METHOD Blink
VAR 
	i : INT;
END_VAR
_toggle(inOffTime:=inBlinkPeriod,inOnTime:=inBlinkPeriod);
_heartBeat := _toggle.IsOn;

FOR i := 0 TO LAST_ICON_INDEX DO
	IF _iconSet[i].BlinkingEnabled AND NOT _iconSet[i].Signal THEN 
		_iconSet[i].SignalBlink := _toggle.IsOn;		
	ELSE
		_iconSet[i].SignalBlink := _iconSet[i].Signal;
	END_IF
END_FOR
END_METHOD

METHOD Clear
_iconSet := _iconSetClear;
_badgeValue := 0;
_currentIndex := 0;
END_METHOD

METHOD CountSignals
VAR
	_iconIndex : INT;
END_VAR
_iconIndex := 0;
_badgeValue := 0;
FOR _iconIndex := 0 TO LAST_ICON_INDEX DO
	IF _iconSet[_iconIndex].Title <> '' AND  _iconSet[_iconIndex].EnableRedIcon THEN 
		_badgeValue := _badgeValue + BOOL_TO_INT(NOT _iconSet[_iconIndex].Signal);
	END_IF
END_FOR
END_METHOD

METHOD SetSignal
VAR_INPUT
	inTitle : STRING;
	inSignal : BOOL;
END_VAR

VAR
	_index : INT;
END_VAR
FOR _index := 0 TO LAST_ICON_INDEX DO 
	IF _iconSet[_index].Title = inTitle THEN 
		_iconSet[_index].Signal := inSignal;
		RETURN;
	END_IF
END_FOR
END_METHOD

END_FUNCTION_BLOCK

// ---- Abstractions/CUBase/Tasks/CUBaseAutomat.TcPOU
FUNCTION_BLOCK ABSTRACT CUBaseAutomat EXTENDS TcoTaskedSequencer
VAR
    _dialog : TcoCore.TcoDialog(THIS^);
    _dialogCustomized : TcoCore.TcoCustomizedDialog(THIS^);
    _dialogWithInput : TcoCore.TcoInputDialog(THIS^);
    {attribute addProperty Name "<#Clear counter#>"}
    _counterDataClear : TcoCore.TcoTask(THIS^);
END_VAR
VAR PERSISTENT
    _counterData : BasicCounterData := (Parent := THIS^);
END_VAR

METHOD PUBLIC ClearCounter
VAR_INPUT
END_VAR
_counterData.Passed := 0;
_counterData.Failed := 0;


_counterData.Total := _counterData.Passed + _counterData.Failed;
END_METHOD

PROPERTY PUBLIC ClearCounterDataTask : REFERENCE TO TcoCore.TcoTask
GET
ClearCounterDataTask ref=_counterDataClear;
END_GET
END_PROPERTY

METHOD Count
VAR_INPUT
	Header 		: EntityHeader;
	
END_VAR


IF NOT Header.IsEmpty THEN

    _counterData.LifeTime := _counterData.LifeTime + 1;

    IF Header.Results.Result = eOverallResult.Failed THEN
        _counterData.Failed := _counterData.Failed + 1;
        _counterData.LifeTimeFailed := _counterData.LifeTimeFailed + 1;
    ELSE
        _counterData.Passed := _counterData.Passed + 1;
        _counterData.LifeTimePassed := _counterData.LifeTimePassed + 1;
    END_IF

END_IF;

_counterData.Total := _counterData.Passed + _counterData.Failed;
END_METHOD

(*~
	<docu>
		<summary>
			Stores the data from this controlled unit into the repository. In addition modifies entity header and controlled unit header.									
		</summary>
	</docu>
~*)
METHOD DataEntityClose
VAR_INPUT
	(*~
	<docu>
		<summary>
			The unique step id definition.
		</summary>			
	</docu>	
	~*)
	inStepID : INT;
	(*~
	<docu>
		<summary>
			If input enum is set to InvokeAndWaitDone  operation will  wait until task reaches the ```Done``` state .
			If input enum is set to InvokeOnly results return True when  task reaches the ```Busy``` state . Later is recomended (neccessary) to check  task  ```Done``` state  , check  task  status.
		</summary>			
	</docu>	
	~*)
	InvokeAction: eDataEntityInvokeType;
END_VAR
VAR_IN_OUT
	Header : CuHeader; 
END_VAR
IF (Step(inStepID,TRUE, 'CLOSE ENTITY DATA')) THEN
    //-------------------------------------		
	IF IsFreshState THEN
		Count(THIS^.StationBase.ProcessDataManager.Data.EntityHeader);
	END_IF
	CASE InvokeAction OF
		eDataEntityInvokeType.InvokeAndWaitDone: 
				StepCompleteWhen(THIS^.StationBase.EntityFlowCloseForOperations(Header).Done);
		eDataEntityInvokeType.InvokeOnly: 
				StepCompleteWhen(THIS^.StationBase.EntityFlowCloseForOperations(Header).Busy);	
	END_CASE;			   		    				
    //-------------------------------------
END_IF
END_METHOD

(*~
	<docu>
		<summary>
			Creates new record in the repository with given EntityId and populates with the current controlled units data.
			In addition modifies entity header and controlled unit header.									
		</summary>
	</docu>
~*)
METHOD DataEntityCreateNew
VAR_INPUT	
	inStepID : INT;
	EntityId : STRING(255);
END_VAR

VAR_IN_OUT
	Header: CuHeader;
END_VAR
IF (Step(inStepID, TRUE, 'CREATE NEW ENTITY DATA')) THEN
    //-------------------------------------		
	StepCompleteWhen(THIS^.StationBase.EntityFlowCreateNew(EntityId, Header).Done);				   		    				
    //-------------------------------------
END_IF
END_METHOD

METHOD DataEntityDiscard
VAR_INPUT	
	inStepID : INT;
	EntityId : STRING(255);
END_VAR
VAR_IN_OUT
	Header: CuHeader;
END_VAR
IF (Step(inStepID, TRUE, 'DISCARD ENTITY DATA')) THEN
    //-------------------------------------		
	StepCompleteWhen(THIS^.StationBase.EntityFlowDiscard(EntityId, Header).Done);				   		    				
    //-------------------------------------
END_IF
END_METHOD

(*~
	<docu>
		<summary>
			Stores data of this controlled unit into the repository.
			In addition modifies entity header and controlled unit header.
			Finalize will set the comprehensive result from InProgress to Passed. 
			If the comprehensive result is Failed the finalizing will not modify the result.									
		</summary>
	</docu>
~*)
METHOD DataEntityFinalize : BOOL
VAR_INPUT
	(*~
	<docu>
		<summary>
			The unique step id definition.
		</summary>			
	</docu>	
	~*)
	inStepID : INT;
	(*~
	<docu>
		<summary>
			If input enum is set to InvokeAndWaitDone  operation will  wait until task reaches the ```Done``` state .
			If input enum is set to InvokeOnly results return True when  task reaches the ```Busy``` state . This option is used when we need to reduce cycle time. Later is recomended (neccessary) to check  task  ```Done``` state  , check  task  status.
		</summary>			
	</docu>	
	~*)
	InvokeAction: eDataEntityInvokeType;
END_VAR
VAR_IN_OUT
	Header: CuHeader;
END_VAR
IF (Step(inStepID,TRUE, 'FINALIZE ENTITY DATA')) THEN
    //-------------------------------------		
		CASE InvokeAction OF
		eDataEntityInvokeType.InvokeAndWaitDone: 
				StepCompleteWhen(THIS^.StationBase.EntityFlowFinalize(Header).Done);
		eDataEntityInvokeType.InvokeOnly: 
				StepCompleteWhen(THIS^.StationBase.EntityFlowFinalize(Header).Busy);	
	END_CASE;			   		    				
		   		    				
    //-------------------------------------
END_IF
END_METHOD

(*~
	<docu>
		<summary>
			Retrieves the data with given EntityId from the repository. In addition modifies entity header and controlled unit header.									
		</summary>
	</docu>
~*)
METHOD DataEntityOpen
VAR_INPUT
	(*~
	<docu>
		<summary>
			The unique step id definition.
		</summary>			
	</docu>	
	~*)
	inStepID : INT;
	(*~
	<docu>
		<summary>
			The definition of jump sptep.Usage of this jump step is when entity does not belong to the Controled unit.
		</summary>			
	</docu>	
	~*)
	inReqStepId: INT;
	inEntityId : STRING(255);
END_VAR
VAR_IN_OUT
	CuHeader: CuHeader;
END_VAR
IF (Step(inStepID, TRUE, 'OPEN ENTITY DATA')) THEN
    //-------------------------------------		
    IF THIS^.StationBase.EntityFlowOpenForOperations(inEntityId, CuHeader).Done THEN
        IF THIS^.StationBase.ProcessDataManager.Data.EntityHeader.IsEmpty THEN
            RequestStep(inReqStepId);
        ELSIF EntityDoesBelong() THEN
            CompleteStep();
        ELSE
            RequestStep(inReqStepId);
        END_IF
    END_IF;
    //-------------------------------------
END_IF
END_METHOD

METHOD EntityDoesBelong : BOOL
VAR_INPUT
END_VAR
EntityDoesBelong:=THIS^.StationBase.ProcessDataManager.Data.EntityHeader.NextStation = THIS^.StationBase.CuId;
END_METHOD

METHOD PUBLIC  HideAllDialogs
VAR_INPUT
END_VAR
_dialog.Restore();
_dialogWithInput.Restore();
_dialogCustomized.Restore();
END_METHOD

METHOD MonitorAnyRecurringFailure
VAR_INPUT
	(*~
	<docu>
		<summary>
			The unique step id definition.
		</summary>			
	</docu>	
	~*)
	inStepID : INT;
	(*~
	<docu>
		<summary>
			The step enable condition.
		</summary>			
	</docu>	
	~*)
	inEnableStep :BOOL;
	inResult : TcoComprehensiveResult;
END_VAR
IF (Step(inStepID,inEnableStep, 'MONITOR ANY RECURRING FAILURE IN SEQUENCE')) THEN
    //-------------------------------------		
	
	IF(inResult.Result<>eOverallResult.Failed ) THEN
		THIS^.StationBase.RecurringFails.AnyRecurringFails.Counter:=0;
		THIS^.StationBase.RecurringFails.AnyRecurringFails.Reached :=FALSE;
		This^.CompleteStep();
	ELSE
		//collect any recurring fails
		IF NOT THIS^.StationBase.RecurringFails.AnyRecurringFails.Reached THEN 
			THIS^.StationBase.RecurringFails.AnyRecurringFails.Counter := THIS^.StationBase.RecurringFails.AnyRecurringFails.Counter +1;
		END_IF
		THIS^.StationBase.RecurringFails.AnyRecurringFails.Reached:=THIS^.StationBase.RecurringFails.AnyRecurringFails.Counter>=THIS^.StationBase._settings.AnyRecurringFailure;
		

		
	

		
		THIS^.Messenger.OnCondition(THIS^.StationBase.RecurringFails.AnyRecurringFails.Reached)
									   .Build()
									   .Append('(Consecutive failure) The number of any recurring failure count has been reached!')
									   .Append(' Failure code: ')
									   .Append(inResult.ErrorCodes)
  									   .Append(' ')
									   .Append(inResult.Failures)						
									   .As()				   
									   .AsError();
									   
		THIS^.StepCompleteWhen(NOT THIS^.StationBase.RecurringFails.AnyRecurringFails.Reached);			
						   
									   
		IF THIS^.StationBase.RecurringFails.AnyRecurringFails.Reached THEN
			
				
			IF(_dialog.Show()
			   .WithCaption('<#(Consecutive failure) The number of any recurring failure count has been reached!#>')
			   .WithText('<#Please acknowledge recurring failure!#>')
			   .WithOk().Answer = TcoCore.eDialogAnswer.OK) THEN
			   
					THIS^.StationBase.RecurringFails.AnyRecurringFails.Counter:=0;
					THIS^.StationBase.RecurringFails.AnyRecurringFails.Reached :=FALSE;
					THIS^.CompleteStep();
			END_IF; 
		END_IF;
	END_IF;
	

	
	
	
 		    				
    //-------------------------------------
END_IF
END_METHOD

METHOD MonitorSameRecurringFailure
VAR_INPUT
	(*~
	<docu>
		<summary>
			The unique step id definition.
		</summary>			
	</docu>	
	~*)
	inStepID : INT;
		(*~
	<docu>
		<summary>
			The step enable condition.
		</summary>			
	</docu>	
	~*)
	inEnableStep :BOOL;
	inResult : TcoComprehensiveResult;
END_VAR
IF (Step(inStepID,inEnableStep, 'MONITOR SAME RECURRING FAILURE IN SEQUENCE')) THEN
    //-------------------------------------		
	
	IF(inResult.Result<>eOverallResult.Failed ) THEN
		THIS^.StationBase.RecurringFails.SameRecurringFails.Counter:=0;
		THIS^.StationBase.RecurringFails.SameRecurringFails.Reached :=FALSE;
		THIS^.CompleteStep();
	ELSE
	
		//collect same recurring
		IF NOT THIS^.StationBase.RecurringFails.SameRecurringFails.Reached THEN 
			IF THIS^.StationBase.RecurringFails.SameRecurringFails.Result.ErrorCodes = inResult.ErrorCodes AND inResult.ErrorCodes <>';' THEN //if error code not defined ignore
				THIS^.StationBase.RecurringFails.SameRecurringFails.Counter := THIS^.StationBase.RecurringFails.SameRecurringFails.Counter +1;
			END_IF;
			THIS^.StationBase.RecurringFails.SameRecurringFails.Result.ErrorCodes := inResult.ErrorCodes ;
		END_IF;
		
		THIS^.StationBase.RecurringFails.SameRecurringFails.Reached:=THIS^.StationBase.RecurringFails.SameRecurringFails.Counter>=THIS^.StationBase._settings.SameRecurringFailure;

			
		THIS^.Messenger.OnCondition(THIS^.StationBase.RecurringFails.SameRecurringFails.Reached)
									   .Build()
									   .Append('(Consecutive failure) The number of same recurring failure count has been reached!')
									   .Append(' Failure code: ')
									   .Append(inResult.ErrorCodes)
  									   .Append(' ')
									   .Append(inResult.Failures)									   									   
									   .As()				   
									   .AsError();
		
		THIS^.StepCompleteWhen(NOT THIS^.StationBase.RecurringFails.SameRecurringFails.Reached);
	

									   
		IF THIS^.StationBase.RecurringFails.SameRecurringFails.Reached THEN
			IF(_dialog.Show()
			   .WithCaption('<#(Consecutive failure) The number of same recurring failure count has been reached!#>')
			   .WithText('<#Please acknowledge recurring failure!#>')
			   .WithOk().Answer = TcoCore.eDialogAnswer.Ok) THEN
			   
					THIS^.StationBase.RecurringFails.SameRecurringFails.Counter:=0;
					THIS^.StationBase.RecurringFails.SameRecurringFails.Reached :=FALSE;
					THIS^.CompleteStep();
			END_IF; 
		END_IF
	END_IF;
	

	
	
	
 		    				
    //-------------------------------------
END_IF
END_METHOD

PROPERTY StationBase : REFERENCE TO CuBase
GET
VAR
    _station : POINTER TO CUBase;
END_VAR
IF __QUERYPOINTER(Parent, _station) THEN // Check if _Parent is Station001
    StationBase REF= _station^;              // If the check is successful dereference a pointer. simlar to THIS^ or SUPER^
END_IF
END_GET
END_PROPERTY

END_FUNCTION_BLOCK

// ---- Abstractions/TcoCore/TcoTaskedSequencer.TcPOU
FUNCTION_BLOCK PUBLIC ABSTRACT TcoTaskedSequencer EXTENDS TcoCore.TcoSequencerBase
VAR
	{attribute addProperty Name "|[[1]AttributeName]|"}
	{attribute addProperty ToolTip "|[[1]AttributeToolTip]|"}
    _task : TcoInnerTask(THIS^);
    _o    : TcoCore.TcoSequencerObserver(THIS^);	
	
	{attribute addProperty Name "|[[1]Cycle Time Analitics]|"} 
	_cycleTimeAnalitics:CycleTimeAnalitics;	
	_startCleanCycleTime: TIME;
	_stopCleanCycleTime: TIME;
	_timer_1: TON;
	_timer_2: TON;
	_detectStartSeq : R_TRIG;

	_customObserver:TcoCustomSequencerObserver(THIS^);
END_VAR

Run();

PROPERTY PUBLIC AverageCleanCycleTime : TIME
GET
AverageCleanCycleTime:=_cycleTimeAnalitics.AverageCleanCycle;
END_GET
END_PROPERTY

PROPERTY PUBLIC AverageCycleTime : TIME
GET
AverageCycleTime:=_cycleTimeAnalitics.Average;
END_GET
END_PROPERTY

(*~
	<docu>
		<summary>
			Completes the actually running step, when the `inCondition` parameter is `TRUE`.
			Method is typically called inside a step as the transition method.
		</summary>			
	</docu>	
~*)
METHOD PROTECTED FINAL Await
VAR_INPUT
    (*~
	<docu>
		<summary>
			The condition under which the step is completed.
		</summary>			
	</docu>	
~*)
    inCondition : BOOL;
END_VAR
i_StepCompleteWhen(inCondition := inCondition);
END_METHOD

(*~
	<docu>
		<summary>
			<para>
				Completes the sequencer, and return the sequencer pointer to the first step in the seuqence.
				Method is typically called inside the last step of the sequence.
			</para>
		</summary>			
	</docu>	
~*)
METHOD PROTECTED FINAL CompleteSequence



i_CompleteSequence();

IF _cycleTimeAnalitics.FilterConstant = 0 THEN;
	_cycleTimeAnalitics.FilterConstant:=10;
END_IF;


IF _cycleTimeAnalitics.Average = T#0S THEN
	_cycleTimeAnalitics.Average:=_SequenceElapsedTime;
END_IF
_cycleTimeAnalitics.Average:= (((_cycleTimeAnalitics.FilterConstant-1)*_cycleTimeAnalitics.Average)+_LastCycleTime)/_cycleTimeAnalitics.FilterConstant;

_startCleanCycleTime:=T#0S;
_stopCleanCycleTime:=T#0S;
END_METHOD

(*~
	<docu>
		<summary>
			Completes the execution of the current step and moves the sequencer pointer to the next step in order of execution.
			The call returns `ITcoObjectRestorer` that allows to restore object upon step completition.
		</summary>		
		<returns></returns>	
	</docu>	
~*)
METHOD PROTECTED FINAL CompleteStep : ITcoObjectRestorer

CompleteStep := i_CompleteStep();
END_METHOD

PROPERTY CustomObserver : REFERENCE TO TcoCustomSequencerObserver
GET
CustomObserver ref= _customObserver;
END_GET
END_PROPERTY

PROPERTY PUBLIC CycleTimeFilterConstant : UINT
GET
CycleTimeFilterConstant:=_cycleTimeAnalitics.FilterConstant;
END_GET
SET // PUBLIC
_cycleTimeAnalitics.FilterConstant:=CycleTimeFilterConstant;
END_SET
END_PROPERTY

(*~
	<docu>
		<summary>
			Main method of the sequener. Custom code needs to be placed here. The sequencer is executed by call of **Instance.Run()** method.
			This method is abstract, and it must be overridden in derived block.
		</summary>
	</docu>
~*)
METHOD PROTECTED  Main : BOOL
END_METHOD

(*~
	<docu>
		<summary>
			Completes the execution of the current step and moves the sequencer pointer to the next step in order of execution.
			The call returns `ITcoObjectRestorer` that allows to restore object upon step completition.
		</summary>		
		<returns></returns>	
	</docu>	
~*)
METHOD PROTECTED FINAL Next : ITcoObjectRestorer
Next := i_CompleteStep();
END_METHOD

METHOD PUBLIC OnAbort : BOOL
SUPER^.Restore();
END_METHOD

METHOD PUBLIC OnDone : BOOL
END_METHOD

METHOD PUBLIC OnError : BOOL
END_METHOD


(*~
	<docu>
		<summary>
			This method is called on sequence completion (the sequencer's last step was completed). 
			This method can be overridden in derived block with a custom logic.
		</summary>			
	</docu>	
~*)
METHOD PROTECTED OnSequenceCompleted
SUPER^.OnSequenceCompleted();
_customObserver.DefineEndTime(Context.RealTimeClock.NowLocalAsTIMESTRUCT());
_customObserver.CompleteSequence();
END_METHOD

METHOD PUBLIC OnStart
_startCleanCycleTime:=T#0S;
_stopCleanCycleTime:=T#0S;
END_METHOD

(*~
	<docu>
		<summary>
			This method is executed upon step completion.
			This method can be overridden in derived block by custom logic.
		</summary>			
	</docu>	
~*)
METHOD PROTECTED OnStepCompleted


_customObserver.Observe(
	inID:= _currentStep.ID, 
	inDescription:= _currentStep.Description, 
	inDuration:= _currentStep.Duration);
END_METHOD

METHOD pr_Close
VAR_INPUT
END_VAR
_lastClosingCycle := Context.StartCycleCount;

IF _sequencerHasError THEN
    OnSequencerError(_sequencerErrorId);
END_IF

_previousNumberOfStepsInSequence := _numberOfStepsInSequence;
Context.Environment.Messaging.Suspend();

IF _modeController._stepIn.Done THEN
    _modeController._stepIn.Restore();
END_IF

Context.Environment.Messaging.Resume();

_restoringSequence := FALSE;
END_METHOD

METHOD pr_Open
VAR
    _message : STRING(255);
END_VAR
_theOrderOfTheCurrentlyEvaluatedStep := 0;

IF _requestStepActive AND
    _requestedStepId <> (MinStepID - 1) AND
    (_modeController.Mode <> eSequencerMode.StepMode OR _modeController._stepIn.Busy OR _checkStepIdRequestedInStepMode) THEN
    _requestStepCycle := _requestStepCycle + 1;
ELSE
    _requestStepCycle := 0;

END_IF

IF _requestStepCycle > 1 AND NOT _sequencerHasError THEN
    _sequencerErrorId        := eSequencerError.StepWithRequestedIdDoesNotExists;
    _message                 := CONCAT('REQUESTED STEP_ID: ', INT_TO_STRING(_requestedStepId));
    _message                 := CONCAT(_message, ' DOES NOT EXIST');
    _currentStep.Description := _message;
    _currentStep.Status      := eStepStatus.Error;
    THIS^.Messenger.Post(_message, eMessageCategory.ProgrammingError);
    _sequencerHasError := TRUE;

END_IF

IF _StepIdUniquenessControlState = eStepIdUniquenessControlState.NotYetStarted OR
    _StepIdUniquenessControlState = eStepIdUniquenessControlState.Requested THEN
    _StepIdUniquenessControlState := eStepIdUniquenessControlState.Started;

END_IF;

_restoringSequence := FALSE;

_lastOpeningCycle := Context.StartCycleCount;
END_METHOD

(*~
	<docu>
		<summary>
			Terminates the currently executed step and set the sequencer's pointer to the step with Id that corresponds to ```inRequestedStepID``` parameter.
			When the order of the requested step is higher than the order of the currently finished step (the requested step is "after" the current one)
			the requested step is started in the same context cycle.
			When the order of the requested step is lower than the order of the currently finished step (the requested step is "before" the current one)
			the requested step is started in the next context cycle.
			If the requested step is not found even in the next context cycle, the sequencer enters error state ```StepWithRequestedIdDoesNotExists```.
			<para>
				See <see cref="TcoCore.eSequencerError"/> for detailed description.
			</para>
		</summary>
	</docu>
~*)
METHOD PROTECTED FINAL RequestRestoreOrigin : ITcoSequencer

VAR
    _message : STRING(254);
END_VAR
RequestRestoreOrigin := i_RequestStep(inRequestedStepID := RESTORE_STEP_ID);
END_METHOD

(*~
	<docu>
		<summary>
			Terminates the currently executed step and set the sequencer's pointer to the step with Id that corresponds to ```inRequestedStepID``` parameter.
			When the order of the requested step is higher than the order of the currently finished step (the requested step is "after" the current one)
			the requested step is started in the same context cycle.
			When the order of the requested step is lower than the order of the currently finished step (the requested step is "before" the current one)
			the requested step is started in the next context cycle.
			If the requested step is not found even in the next context cycle, the sequencer enters error state ```StepWithRequestedIdDoesNotExists```.
			<para>
				See <see cref="TcoCore.eSequencerError"/> for detailed description.
			</para>
		</summary>
	</docu>
~*)
METHOD PROTECTED FINAL RequestStep : ITcoSequencer
VAR_INPUT
    (*~
		<docu>
			<summary>
				StepId of the step to be executed.
			</summary>
		</docu>
	~*)
    inRequestedStepID : INT := MinStepID - 1;
END_VAR
VAR
    _message : STRING(254);
END_VAR
RequestStep := i_RequestStep(inRequestedStepID := inRequestedStepID);
END_METHOD

(*~
	<docu>
		<summary>
			This method resets the sequencer cycle time . 
				Method is typically called before starting the sequence(e.g.in ground position task) .
		</summary>		
		<returns></returns>	
	</docu>	
~*)
METHOD PUBLIC ResetCycleTime
VAR_INPUT
END_VAR

_cycleTimeAnalitics.Average:=T#0S;
_cycleTimeAnalitics.AverageCleanCycle:=T#0S;
END_METHOD

METHOD PRIVATE ResetTimers
VAR_INPUT
END_VAR
_timer_1.IN:=FALSE;
_timer_2.IN:=FALSE;
END_METHOD

(*~
	<docu>
		<summary>
			<para>
				This method resets the sequencer. 
				Method is typically called before starting the sequence or after error has occured in the sequence.
			</para>
		</summary>			
	</docu>	
~*)
METHOD PUBLIC Restore : ITcoRestorable
SUPER^.Restore();
Task.Restore();
END_METHOD

(*~
	<docu>
		<summary>
			<para>
				Ensures calling the Open(), Main() and Close() methods in the desired order.
				This method is final, so it cannot be overloaded. The **Instance.Run()** needs to be called cyclically inside the appropriate context.
			</para>
		</summary>			
	</docu>	
~*)
METHOD PUBLIC FINAL Run
VAR
    _message : STRING;
END_VAR
IF (_task.Execute()) THEN
    THIS^.pr_Open();

    THIS^.Observer := _o;
    THIS^.Main();
	_detectStartSeq(CLK:=_cycleTimer.ET > T#0S);
    IF _detectStartSeq.Q THEN
        CustomObserver.Clear();
        CustomObserver.DefineStartTime(Context.RealTimeClock.NowLocalAsTIMESTRUCT());
    END_IF

    _customObserver();
    THIS^.pr_Close();
END_IF;
END_METHOD

(*~
	<docu>
		<summary>
			This method s used to start the clean cycle time measurement . 
				Method is typically called at the beggining of the sequence(e.g.in automat sequence) .
		</summary>		
		<returns></returns>	
	</docu>	
~*)

METHOD PUBLIC StartCleanCycleTime
VAR_INPUT
END_VAR
_stopCleanCycleTime:=t#0s;
_startCleanCycleTime:=_SequenceElapsedTime;
END_METHOD

METHOD PROTECTED Step : BOOL
VAR_INPUT
    (*~
	<docu>
		<summary>
			StepId of the current step.
			<remarks>			
				<note type="important">
					This number must be unique throughout the complete sequence.
					It must be a constant or numerical literal and it must not change during the life-time of the sequencer. 
				</note>
			</remarks>
		</summary>		
	</docu>	
~*)
    inStepID : INT;
    (*~
	<docu>
		<summary>
			If this value is false, step body is not executed and execution is moved to the next enabled step.
		</summary>				
	</docu>	
~*)
    inEnabled : BOOL;
    (*~
	<docu>
		<summary>
			Step description text.
		</summary>				
	</docu>	
~*)
    inStepDescription : STRING(254);
END_VAR
Step := i_Step(inStepID := inStepID, inEnabled := inEnabled, inStepDescription := inStepDescription);
END_METHOD

(*~
	<docu>
		<summary>
			Completes the actually running step, when the `inCondition` parameter is `TRUE`.
			Method is typically called inside a step as the transition method.
		</summary>			
	</docu>	
~*)
METHOD PROTECTED FINAL StepCompleteWhen
VAR_INPUT
    (*~
	<docu>
		<summary>
			The condition under which the step is completed.
		</summary>			
	</docu>	
~*)
    inCondition : BOOL;
END_VAR
i_StepCompleteWhen(inCondition := inCondition);
END_METHOD

(*~
	<docu>
		<summary>
			This method s used to stop the clean cycle time measurement . 
				Method is typically called at the end of the sequence(e.g.in automat sequence )  .
		</summary>		
		<returns></returns>	
	</docu>	
~*)

METHOD PUBLIC StopCleanCycleTime
VAR_INPUT
END_VAR

VAR
	cleanCycleTime: TIME;
END_VAR
_stopCleanCycleTime:=_SequenceElapsedTime;

cleanCycleTime:=T#0S;
IF _stopCleanCycleTime>_startCleanCycleTime THEN
	cleanCycleTime:=_stopCleanCycleTime-_startCleanCycleTime;
 END_IF;

IF _cycleTimeAnalitics.FilterConstant = 0 THEN;
	_cycleTimeAnalitics.FilterConstant:=10;
END_IF;


IF _cycleTimeAnalitics.AverageCleanCycle = T#0S THEN
	_cycleTimeAnalitics.AverageCleanCycle:=_stopCleanCycleTime;
END_IF
_cycleTimeAnalitics.AverageCleanCycle:= (((_cycleTimeAnalitics.FilterConstant-1)*_cycleTimeAnalitics.AverageCleanCycle)+cleanCycleTime)/_cycleTimeAnalitics.FilterConstant;
END_METHOD

PROPERTY Task : REFERENCE TO TcoTask
GET
Task REF= _task;
END_GET
END_PROPERTY

METHOD PUBLIC FINAL Timer_1 : BOOL
VAR_INPUT
	Condition : BOOL;
	PT : TIME;
END_VAR
_timer_1(IN:= Condition  and  not IsFreshState, PT:=PT);
Timer_1 := _timer_1.Q;
END_METHOD

METHOD PUBLIC FINAL Timer_2 : BOOL
VAR_INPUT
	Condition : BOOL;
	PT : TIME;
END_VAR
_timer_2(IN:= Condition and not IsFreshState, PT:=PT);
Timer_2 := _timer_2.Q;
END_METHOD

END_FUNCTION_BLOCK

// ---- Abstractions/TcoCore/TcoCustomSequencerObserver.TcPOU
FUNCTION_BLOCK TcoCustomSequencerObserver EXTENDS TcoObject 
VAR
	//~
    _data            : TcoCustomExportSeqData;
	//~
	_dataToExport            : TcoCustomExportSeqData;
	

	_exportSeqData:TcoCore.TcoRemoteTask(THIS^);
	_order:UINT;
END_VAR

VAR CONSTANT
    MAX_STEPS : UINT := 150;
END_VAR

_exportSeqData();

{attribute 'hide'}
METHOD Clear : BOOL
VAR 
	i : INT;
	blank : TcoCustomStepDetails;
END_VAR
{warning disable C0196}
FOR i := 0 TO MAX_STEPS DO
{warning enable C0196}
	_data.Steps[i] := blank;	
END_FOR
_order:=0;
END_METHOD

METHOD CompleteSequence
VAR_INPUT
END_VAR

_dataToExport:=_data;

IF _exportSeqData._isInitialized  THEN
	
	_exportSeqData.Restore();
	_exportSeqData.Invoke();
  
	
END_IF
END_METHOD

METHOD DefineControledUnit
VAR_INPUT
	inCuid: UINT;
END_VAR
_data.CuId:=inCuid;
END_METHOD

METHOD DefineEndTime
VAR_INPUT
	inTime:Tc2_Utilities.TIMESTRUCT;
END_VAR
_data.EndTime.Year :=  inTime.wYear;
_data.EndTime.Month :=  inTime.wMonth;
_data.endTime.Day :=  inTime.wDay;
_data.endTime.Hour :=  inTime.wHour;
_data.endTime.Minute :=  inTime.wMinute;
_data.endTime.Second :=  inTime.wSecond;
_data.endTime.Milliseconds :=  inTime.wMilliseconds;
END_METHOD

METHOD DefineStartTime
VAR_INPUT
	inTime:Tc2_Utilities.TIMESTRUCT;
END_VAR
_data.startTime.Year :=  inTime.wYear;
_data.startTime.Month :=  inTime.wMonth;
_data.startTime.Day :=  inTime.wDay;
_data.startTime.Hour :=  inTime.wHour;
_data.startTime.Minute :=  inTime.wMinute;
_data.startTime.Second :=  inTime.wSecond;
_data.startTime.Milliseconds :=  inTime.wMilliseconds;
END_METHOD

PROPERTY ExportSeqData : REFERENCE TO TcoCore.TcoRemoteTask
GET
ExportSeqData ref=_exportSeqData;
END_GET
END_PROPERTY

(*~
	<docu>
		<summary>
			Provides the mechanism to observe steps in the sequence and to gather basic infomation about step status and perfomance.
		</summary>			
	</docu>	
~*)
METHOD Observe
VAR_INPUT
	
	(*~
	<docu>
		<summary>
			Step identification number.
		</summary>	
		<remarks>			
 			<note type="important">
				This number must be unique throughout the complete sequence. It is required to uniquely identify the step of the sequence.
			</note>
			<para>
				The <see cref="PlcDocu.TcoCore.TcoSequencer.RequestStep"/> method is using this number to jump to the required step.
			</para>
		</remarks>
	</docu>	
	~*)
		{attribute addProperty Name "<#Step ID#>"}
		inID: INT;


	(*~
		<docu>
			<summary>
				Step description text.
			</summary>				
		</docu>	
	~*)
		{attribute addProperty Name "<#Step description#>"}
		inDescription: STRING(254);

	(*~
		<docu>
			<summary>
				Step duration time.
			</summary>				
		</docu>	
	~*)	
		{attribute addProperty Name "<#Step duration#>"}
		inDuration : TIME;	


END_VAR

VAR
	_timeStruct: Tc2_Utilities.TIMESTRUCT;
END_VAR

IF(_order <= MAX_STEPS)  THEN
	_data.Steps[_order].ID := inID;
	_data.Steps[_order].Description := inDescription;
	_data.Steps[_order].Duration := inDuration;
	_timeStruct:=Context.RealTimeClock.NowLocalAsTIMESTRUCT();
	
	_data.Steps[_order].TimeStamp.Year :=  _timeStruct.wYear;
	_data.Steps[_order].TimeStamp.Month :=  _timeStruct.wMonth;
	_data.Steps[_order].TimeStamp.Day :=  _timeStruct.wDay;
	_data.Steps[_order].TimeStamp.Hour :=  _timeStruct.wHour;
	_data.Steps[_order].TimeStamp.Minute :=  _timeStruct.wMinute;
	_data.Steps[_order].TimeStamp.Second :=  _timeStruct.wSecond;
	_data.Steps[_order].TimeStamp.Milliseconds :=  _timeStruct.wMilliseconds;


		
	
	_order:=_order+1;
END_IF;
END_METHOD

METHOD SetCycleId
VAR_INPUT
	inId:string(254);
END_VAR
_data.CycleId:=inId;
END_METHOD

END_FUNCTION_BLOCK

// ---- Abstractions/Generic/LightTower/TcoLightTower.TcPOU
FUNCTION_BLOCK TcoLightTower EXTENDS TcoCore.TcoComponent
VAR_IN_OUT
	{attribute clr [RenderIgnore()]}
	inoGreenLight   :  BOOL;
	
	{attribute clr [RenderIgnore()]}
	inoRedLight     :  BOOL;
	
	{attribute clr [RenderIgnore()]}
	inoOrangeLight  :  BOOL;
	
	{attribute clr [RenderIgnore()]}
	inoBlueLight    :  BOOL;

	{attribute clr [RenderIgnore()]}
	inoHorn         :  BOOL;
END_VAR

VAR
	
	
	{attribute addProperty Name "<#Status#>"}
    {attribute clr [ReadOnly()]}
    _status : TcoLightTower_Status;

	{attribute addProperty Name "<#Config#>"}
    _config : TcoLightTower_Config;
	
    _materrialError : bool;

	//~
	_controlledUnits      : ARRAY [0..12] OF ICUBase;
	//~			
	
	
	// group states

	//~
	{attribute clr [RenderIgnore()]}
	_blinker              : TcoUtilities.TcoBlinker(THIS^);
	{attribute clr [RenderIgnore()]}
	_blinkerSlow              : TcoUtilities.TcoBlinker(THIS^);
	//~

END_VAR

IF _controlledUnits[0] = 0 THEN
    THIS^.Messenger.Programming('<#Missing link to Controlled unit! No function is being executed!#>');
    RETURN;
END_IF

inoGreenLight := FALSE;
inoRedLight := FALSE;
inoOrangeLight := FALSE;
inoBlueLight := FALSE;
inoHorn := FALSE;

_blinker(inOffTime := T#500MS, inOnTime := T#500MS); //2 Hz
_blinkerSlow(inOffTime := T#1250MS, inOnTime := T#1250MS); //0.8 Hz

THIS^.Initialize();

//ground
IF _status.State.AnyGrounding THEN
    inoGreenLight := _blinker.IsOn;
    inoRedLight := _status.State.AnyInError AND _blinker.IsOn;
    inoOrangeLight := _status.State.AnyInWarning AND _blinker.IsOn;
END_IF

//auto
IF _status.State.AllInAuto AND NOT _status.State.AnyInStepMode AND NOT _status.State.AnyInError AND _status.State.AnyInWarning THEN
    inoGreenLight := TRUE; // ok production
ELSIF _status.State.AllInAuto AND _status.State.AnyInStepMode THEN
    inoGreenLight := _blinker.IsOn; //step mode
ELSIF _status.State.AllInAuto AND NOT _status.State.AnyInStepMode THEN
    inoGreenLight := TRUE; // ok production
    inoRedLight := _status.State.AnyInError AND _blinker.IsOn;
    inoOrangeLight := _status.State.AnyInWarning AND _blinker.IsOn;
ELSIF _status.State.AllInManual  THEN

    inoOrangeLight :=  _blinker.IsOn;

END_IF;

IF NOT _config.HornEnabled THEN
    inoHorn := FALSE;
END_IF;

//todo blue should be suitable for material feeding
IF _materrialError AND _status.State.AllInAuto THEN
	inoBlueLight :=  _blinker.IsOn;
END_IF

METHOD AddControlledUnit : BOOL
VAR_INPUT
 	inControlledUnit : ICUBase;
END_VAR
VAR
	i : UINT;
END_VAR
AddControlledUnit := FALSE;

IF inControlledUnit = 0 THEN
	RETURN;
END_IF

FOR i := 0 TO _config.MaxControledUnits DO
	IF _controlledUnits[i] = inControlledUnit THEN
		AddControlledUnit := TRUE;
		RETURN;
	END_IF
	
	IF 	_controlledUnits[i] = 0 THEN
		_controlledUnits[i] := inControlledUnit;
		AddControlledUnit    := TRUE;
		RETURN;
	END_IF
END_FOR
END_METHOD

PROPERTY Config :REFERENCE TO TcoLightTower_Config
GET
Config ref=_config;
END_GET
END_PROPERTY

METHOD Initialize : BOOL
VAR
	i : UINT;

END_VAR
_status.State.AllInAuto := TRUE;
_status.State.AllInGrounding := TRUE;
_status.State.AllInManual := TRUE;
_status.State.AllIdle := TRUE;
_status.State.AllGrounded := TRUE;
_status.State.AllInStepMode := TRUE;
_status.State.AllSuspended := TRUE;
_status.State.AllRecovered := TRUE;
_status.State.AllInactiveOrManualOrGrounded :=true;
_status.State.AnyInAuto := FALSE;
_status.State.AnyInManual := FALSE;
_status.State.AnyGrounding := FALSE;
_status.State.AnyInStepMode := FALSE;

_status.State.AnyInWarning := FALSE;
_status.State.AnyInError := FALSE;

i := 0;

FOR i := 0 TO _config.MaxControledUnits DO
    IF _controlledUnits[i] <> 0 THEN
        _status.State.AllInAuto := _status.State.AllInAuto AND _controlledUnits[i].StatusInfo.Mode = eCUMode.AutomatMode;
        _status.State.AllInManual := _status.State.AllInManual AND _controlledUnits[i].StatusInfo.Mode = eCUMode.ManualMode;
        _status.State.AllIdle := _status.State.AllIdle AND _controlledUnits[i].StatusInfo.Mode = eCUMode.NoMode;
        _status.State.AllInGrounding := _status.State.AllInGrounding AND
            (_controlledUnits[i].StatusInfo.Mode = eCUMode.GroundModeDone XOR
            _controlledUnits[i].StatusInfo.Mode = eCUMode.GroundMode);
        _status.State.AllGrounded := _status.State.AllGrounded AND _controlledUnits[i].StatusInfo.Mode = eCUMode.GroundModeDone;
        _status.State.AllInStepMode := _status.State.AllInStepMode AND _controlledUnits[i].StatusInfo.CurrentIsInStepMode;
        _status.State.AllSuspended := _status.State.AllSuspended AND _controlledUnits[i].SuspendTask.Task.Done;
		_status.State.AllRecovered := _status.State.AllRecovered AND _controlledUnits[i].RecoverTask.Task.Done;
		_status.State.AllInactiveOrManualOrGrounded := _status.State.AllInactiveOrManualOrGrounded 
											AND (_controlledUnits[i].StatusInfo.Mode = eCUMode.ManualMode 
												OR _controlledUnits[i].StatusInfo.Mode = eCUMode.NoMode 
												OR _controlledUnits[i].StatusInfo.Mode = eCUMode.GroundModeDone );
		
        _status.State.AnyInAuto := _status.State.AnyInAuto OR _controlledUnits[i].StatusInfo.Mode = eCUMode.AutomatMode;
        _status.State.AnyInManual := _status.State.AnyInManual OR _controlledUnits[i].StatusInfo.Mode = eCUMode.ManualMode;
        _status.State.AnyInStepMode := _status.State.AnyInStepMode OR _controlledUnits[i].StatusInfo.CurrentIsInStepMode;
        _status.State.AnyGrounding := _status.State.AnyGrounding OR
            (_controlledUnits[i].StatusInfo.Mode = eCUMode.GroundModeDone OR
            _controlledUnits[i].StatusInfo.Mode = eCUMode.GroundMode);
		_status.State.AnyInWarning := _status.State.AnyInWarning OR _controlledUnits[i].StatusInfo.State =eCUState.HasWarning;	
		_status.State.AnyInError := _status.State.AnyInError  OR _controlledUnits[i].StatusInfo.State =eCUState.HasError;	
	

    ELSE
        EXIT;
    END_IF
END_FOR
END_METHOD

PROPERTY PUBLIC MaterialError : Reference to BOOL
GET
MaterialError ref=_materrialError;
END_GET
END_PROPERTY

METHOD Restore :  TcoCore.ITcoRestorable
VAR
	i : UINT;
END_VAR
// clear all linked Controlled units
FOR i := 0 TO _config.MaxControledUnits DO
	_controlledUnits[i] := 0;
END_FOR



THIS^.Messenger.UnPin();
END_METHOD

(*~
	<docu>
		<summary>
		    Custom service (manual, maintenance) logic.
			This method must be implemented in derived class.
		</summary>			
	</docu>	
~*)
METHOD PROTECTED  ServiceMode
END_METHOD

PROPERTY Status : REFERENCE TO TcoLightTower_Status
GET
Status REF=_status;
END_GET
END_PROPERTY

END_FUNCTION_BLOCK

// ---- Abstractions/Safety/ControlledZone/TcoControlledZone.TcPOU
FUNCTION_BLOCK TcoControlledZone EXTENDS TcoCore.TcoComponent
VAR_INPUT
    {attribute clr [RenderIgnore()]}
    inDoorCircuit : ITcoDoorCircuit;

    {attribute clr [RenderIgnore()]}
    inAirPressureOK : BOOL;

    //	{attribute clr [RenderIgnore()]}
    //	inEstopActive		      : BOOL;

END_VAR

VAR

    {attribute addProperty Name "<#Status#>"}
    {attribute clr [ReadOnly()]}
    _status : TcoControlledZone_Status;

    {attribute addProperty Name "<#Config#>"}
    _config : TcoControlledZone_Config;

   //~
    _controlledUnits : ARRAY[0..12] OF ICUBase;

    {attribute clr [RenderIgnore()]}
    _controlButtons : ARRAY[0..4] OF ITcoControlButtons;

    {attribute clr [RenderIgnore()]}
    _controlKeyMode : ARRAY[0..2] OF ITcoKeyMode;

    {attribute clr [RenderIgnore()]}
    _controlKeyNormalService : ARRAY[0..2] OF ITcoKeyNormalSevice;
	//~
    // group states

    //~
    _blinker : TcoUtilities.TcoBlinker(THIS^);
    {attribute clr [CompilerOmits("BuilderPlainer", "BuilderOnliner","BuilderOnlinerInterface","BuilderShadowerInterface")]}
    _blinkerSlow : TcoUtilities.TcoBlinker(THIS^);
	//~
    {attribute addProperty Name "<#Ground task#>"}
    _groundTask : TcoControlledZoneActionTask(THIS^);
    {attribute addProperty Name "<#Automat task#>"}
    _autoTask : TcoControlledZoneActionTask(THIS^);

    {attribute addProperty Name "<#Recover task#>"}
    _recoverTask : TcoControlledZoneActionTask(THIS^);

    {attribute addProperty Name "<#Suspend task#>"}
    _suspendTask : TcoControlledZoneActionTask(THIS^);

    {attribute addProperty Name "<#Key Auto task#>"}
    _keyAutoTask : TcoControlledZoneActionTask(THIS^);

    {attribute addProperty Name "<#Key Manual task#>"}
    _keyManualTask : TcoControlledZoneActionTask(THIS^);

    {attribute addProperty Name "<#Key Step task#>"}
    _keyStepTask : TcoControlledZoneActionTask(THIS^);

    {attribute addProperty Name "<#Key service task#>"}
    _keyServiceTask : TcoControlledZoneActionTask(THIS^);

    {attribute clr [RenderIgnore()]}
    _timerDoorsLocked : TON;
    {attribute clr [RenderIgnore()]}
    _timerAirPressureMonitor : TON;

    {attribute clr [RenderIgnore()]}
    _serviceKeyRising : R_Trig;

    {attribute clr [RenderIgnore()]}
    _serviceKeyFalling : F_Trig;

    {attribute clr [RenderIgnore()]}
    _recoverTaskInvokeFalling : F_Trig;

    {attribute clr [RenderIgnore()]}
    _suspendTaskInvokeFalling : F_Trig;

    {attribute clr [RenderIgnore()]}
    _recoverTaskInvokeRising : R_Trig;

    {attribute clr [RenderIgnore()]}
    _suspendTaskInvokeRising : R_Trig;

    {attribute clr [RenderIgnore()]}
    _groundTaskInvokeFalling : F_Trig;

    {attribute clr [RenderIgnore()]}
    _autoTaskInvokeFalling : F_Trig;

    {attribute clr [RenderIgnore()]}
    _groundTaskInvokeRising : F_Trig;

    {attribute clr [RenderIgnore()]}
    _autoTaskInvokeRising : F_Trig;

    {attribute clr [RenderIgnore()]}
    _keyAutoTaskInvokeFalling : F_Trig;
    {attribute clr [RenderIgnore()]}
    _keyAutoTaskInvokeRising : R_Trig;

    {attribute clr [RenderIgnore()]}
    _keyManualTaskInvokeFalling : F_Trig;
    {attribute clr [RenderIgnore()]}
    _keyManualTaskInvokeRising : R_Trig;

    {attribute clr [RenderIgnore()]}
    _keyStepTaskInvokeFalling : F_Trig;
    {attribute clr [RenderIgnore()]}
    _keyStepTaskInvokeRising : R_Trig;

    {attribute clr [RenderIgnore()]}
    _keyServiceTaskInvokeFalling : F_Trig;
    {attribute clr [RenderIgnore()]}
    _keyServiceTaskInvokeRising : R_Trig;
	
		
    _airPressureOk : BOOL;
    _conditionToRunAreSufficient : BOOL;
	//~
	cu: INT;
	//~
END_VAR

IF _controlledUnits[0] = 0 THEN
    THIS^.Messenger.Programming('<#Missing link to Controlled unit! No function is being executed!#>');
    RETURN;
END_IF

IF _controlButtons[0] = 0 OR _controlKeyMode[0] = 0 OR _controlKeyNormalService[0] = 0 THEN
    THIS^.Messenger.Programming('<#Missing link to control panel components (Buttons, Mode Keys, Normal/Service)! No function is being executed!#>');
    RETURN;
END_IF

_blinker(inOffTime := T#500MS, inOnTime := T#500MS); //2 Hz
_blinkerSlow(inOffTime := T#1250MS, inOnTime := T#1250MS); //0.8 Hz

THIS^.Initialize();

//presure monitoring
_airPressureOk := TRUE;
_timerAirPressureMonitor(IN := NOT inAirPressureOK, PT := _config.AirPressureErrorTime);
IF _timerAirPressureMonitor.Q THEN
    _airPressureOk := FALSE;
    THIS^.Messenger.Error('<#Air pressure is not sufficient!#>').Pin();
	
	FOR cu := 0 TO _config.MaxControledUnits DO

        IF _controlledUnits[cu] <> 0 THEN

            _controlledUnits[cu].AutomatTask.Task.Restore();
            _controlledUnits[cu].GroundTask.Task.Restore();
            _controlledUnits[cu].ManualTask.Task.Restore();

        ELSE
            EXIT;
        END_IF
    END_FOR
END_IF;

//Estop monitoring
//IF THIS^.inEstopActive THEN
//    inDoorCircuit.UnLock();
//    THIS^.Messenger.Error('<#Emergency stop active: Unlocking doors!#>').Pin();
//END_IF
// Global Voltage monitoring
IF NOT inDoorCircuit.IsGlobalVoltageOk THEN
    inDoorCircuit.UnLock();
    THIS^.Messenger.Error('<#Global control voltage interrupted: Unlocking doors!#>').Pin();

    FOR cu := 0 TO _config.MaxControledUnits DO

        IF _controlledUnits[cu] <> 0 THEN

            _controlledUnits[cu].AutomatTask.Task.Restore();
            _controlledUnits[cu].GroundTask.Task.Restore();
            _controlledUnits[cu].ManualTask.Task.Restore();

        ELSE
            EXIT;
        END_IF
    END_FOR

END_IF

//Voltage monitoring todo
_timerDoorsLocked(IN := inDoorCircuit.IsClosed AND inDoorCircuit.IsLocked AND inDoorCircuit.IsLocalDoorsVoltageOk, PT := _config.DoorsLocked);

IF _timerDoorsLocked.Q THEN
    IF NOT inDoorCircuit.IsLocalVoltageOk THEN
        // unlock doors in case that control voltage goes down and it shouldn't
        inDoorCircuit.UnLock();
        THIS^.Messenger.Error('<#Local voltage interrupted: Unlocking doors!#>');
		
		FOR cu := 0 TO _config.MaxControledUnits DO

        IF _controlledUnits[cu] <> 0 THEN

            _controlledUnits[cu].AutomatTask.Task.Restore();
            _controlledUnits[cu].GroundTask.Task.Restore();
            _controlledUnits[cu].ManualTask.Task.Restore();

        ELSE
            EXIT;
        END_IF
    END_FOR
    END_IF
END_IF

_conditionToRunAreSufficient := (inAirPressureOK OR _timerAirPressureMonitor.ET < _timerAirPressureMonitor.PT) (*AND NOT inEstopActive*) AND
    inDoorCircuit.IsGlobalVoltageOk AND
    inDoorCircuit.IsLocalVoltageOk;

_recoverTaskInvokeRising(CLK := _status.State.AnyButtonRecover);
_recoverTaskInvokeFalling(CLK := _status.State.AnyButtonRecover);

IF _recoverTaskInvokeRising.Q THEN
    _recoverTask.Restore();
END_IF

IF _recoverTaskInvokeFalling.Q THEN
    _recoverTask.Invoke();
    _suspendTask.Restore();
END_IF

_suspendTaskInvokeRising(CLK := _status.State.AnyButtonSuspend);
_suspendTaskInvokeFalling(CLK := _status.State.AnyButtonSuspend);

IF _suspendTaskInvokeRising.Q THEN
    _suspendTask.Restore();
END_IF

IF _suspendTaskInvokeFalling.Q THEN
    _suspendTask.Invoke();
    _recoverTask.Restore();
END_IF

_groundTaskInvokeRising(CLK := _status.State.AnyButtonGround);

IF _groundTaskInvokeRising.Q THEN
    _groundTask.Restore();
END_IF

_groundTaskInvokeFalling(CLK := _status.State.AnyButtonGround);

IF _groundTaskInvokeFalling.Q THEN
    _groundTask.Invoke();
END_IF

_groundTask.Enabled :=
    (_conditionToRunAreSufficient AND inDoorCircuit.IsLocalDoorsVoltageOk AND _status.State.AllKeysAuto AND _status.State.AllKeysNormal);

IF _groundTask.Busy THEN
    _autoTask.Restore();
END_IF

_autoTaskInvokeRising(CLK := _status.State.AnyButtonAuto);

IF _autoTaskInvokeRising.Q THEN
    _autoTask.Restore();
END_IF

_autoTaskInvokeFalling(CLK := _status.State.AnyButtonAuto);

IF _autoTaskInvokeFalling.Q THEN
    _autoTask.Invoke();
END_IF

_autoTask.Enabled :=
    (_conditionToRunAreSufficient AND inDoorCircuit.IsLocalDoorsVoltageOk AND _status.State.AllKeysAuto AND _status.State.AllKeysNormal);

//----------keys -----------

// key auto
_keyAutoTaskInvokeFalling(CLK := _status.State.AllKeysAuto);
_keyAutoTaskInvokeRising(CLK := _status.State.AllKeysAuto);

IF _keyAutoTaskInvokeRising.Q THEN
    _keyAutoTask.Invoke();
END_IF

IF _keyAutoTaskInvokeFalling.Q THEN
    _keyAutoTask.Restore();
END_IF

// key manual
_keyManualTaskInvokeRising(CLK := _status.State.AnyKeyManual);
_keyManualTaskInvokeFalling(CLK := _status.State.AnyKeyManual);

IF _keyManualTaskInvokeRising.Q THEN
    _keyManualTask.Invoke();
END_IF

IF _keyManualTaskInvokeFalling.Q THEN
    _keyManualTask.Restore();
END_IF

IF _status.State.AnyKeyStep AND _keyStepTask.Ready THEN
    _keyStepTask.Invoke();
END_IF

IF _status.State.AnyKeyStep AND _keyStepTask.Done THEN
    _keyStepTask.Restore();
END_IF

_keyStepTaskInvokeFalling(CLK := _status.State.AnyKeyStep);

IF _keyStepTaskInvokeFalling.Q THEN
    _keyStepTask.Restore();
END_IF

// key service
_keyServiceTaskInvokeRising(CLK := _status.State.AnyKeyService);
_keyServiceTaskInvokeFalling(CLK := _status.State.AnyKeyService);

IF _keyServiceTaskInvokeRising.Q THEN
    _keyServiceTask.Invoke();
END_IF

IF _keyServiceTaskInvokeFalling.Q THEN
    _keyServiceTask.Restore();
END_IF

// Handling of buttons
THIS^.ButtonRecover();
THIS^.ButtonSuspend();
THIS^.ButtonGround();
THIS^.ButtonAuto();

// Handling of key 1
THIS^.KeyAuto();
THIS^.KeyManual();
THIS^.KeyStep();

// Handling of Key Normal/Service
THIS^.KeyService();

METHOD AddControlButtons : BOOL
VAR_INPUT
 	inControlButtons : ITcoControlButtons;
END_VAR
VAR
	i : UINT;
END_VAR
AddControlButtons := FALSE;

IF inControlButtons = 0 THEN
	RETURN;
END_IF

FOR i := 0 TO _config.MaxControlButtons DO
	IF _controlButtons[i] = inControlButtons THEN
		AddControlButtons := TRUE;
		RETURN;
	END_IF
	
	IF 	_controlButtons[i] = 0 THEN
		_controlButtons[i] := inControlButtons;
		AddControlButtons  := TRUE;
		RETURN;
	END_IF
END_FOR
END_METHOD

METHOD AddControlledUnit : BOOL
VAR_INPUT
 	inControlledUnit : ICUBase;
END_VAR
VAR
	i : UINT;
END_VAR
AddControlledUnit := FALSE;

IF inControlledUnit = 0 THEN
	RETURN;
END_IF

FOR i := 0 TO _config.MaxControledUnits DO
	IF _controlledUnits[i] = inControlledUnit THEN
		AddControlledUnit := TRUE;
		RETURN;
	END_IF
	
	IF 	_controlledUnits[i] = 0 THEN
		_controlledUnits[i] := inControlledUnit;
		AddControlledUnit    := TRUE;
		RETURN;
	END_IF
END_FOR
END_METHOD

METHOD AddKeyMode : BOOL
VAR_INPUT
 	inKeyMode : ITcoKeyMode;
END_VAR
VAR
	i : UINT;
END_VAR
AddKeyMode := FALSE;

IF inKeyMode = 0 THEN
	RETURN;
END_IF

FOR i := 0 TO  _config.MaxKeyMode DO
	IF _controlKeyMode[i] = inKeyMode THEN
		AddKeyMode := TRUE;
		RETURN;
	END_IF
	
	IF 	_controlKeyMode[i] = 0 THEN
		_controlKeyMode[i] := inKeyMode;
		AddKeyMode    := TRUE;
		RETURN;
	END_IF
END_FOR
END_METHOD

METHOD AddKeyNormalService : BOOL
VAR_INPUT
 	inKeyNormalService : ITcoKeyNormalSevice;
END_VAR
VAR
	i : UINT;
END_VAR
AddKeyNormalService := FALSE;

IF inKeyNormalService = 0 THEN
	RETURN;
END_IF

FOR i := 0 TO _config.MaxKeyNormalService DO
	IF _controlKeyNormalService[i] = inKeyNormalService THEN
		AddKeyNormalService := TRUE;
		RETURN;
	END_IF
	
	IF 	_controlKeyNormalService[i] = 0 THEN
		_controlKeyNormalService[i] := inKeyNormalService;
		AddKeyNormalService    := TRUE;
		RETURN;
	END_IF
END_FOR
END_METHOD

PROPERTY PUBLIC AirPressureOk : bool
GET
AirPressureOk:=_airPressureOk;
END_GET
END_PROPERTY

{attribute 'monitoring' := 'variable'}
PROPERTY AnyButtonAuto : BOOL
GET
AnyButtonAuto := _status.State.AnyButtonAuto;
END_GET
SET
VAR
	button : UINT;
END_VAR
FOR button := 0 TO _config.MaxControlButtons DO
	IF _controlButtons[button] <> 0 THEN
		_controlButtons[button].ButtonAuto := AnyButtonAuto;
	ELSE
		EXIT;
	END_IF
END_FOR
END_SET
END_PROPERTY

{attribute 'monitoring' := 'variable'}
PROPERTY AnyButtonGround : BOOL
GET
AnyButtonGround := _Status.State.AnyButtonGround;
END_GET
SET
VAR
	button : UINT;
END_VAR
FOR button := 0 TO _config.MaxControlButtons DO
	IF _controlButtons[button] <> 0 THEN
		_controlButtons[button].ButtonGround := AnyButtonGround;
	ELSE
		EXIT;
	END_IF
END_FOR
END_SET
END_PROPERTY

{attribute 'monitoring' := 'variable'}
PROPERTY AnyButtonRecover : BOOL
GET
AnyButtonRecover := _status.State.AnyButtonRecover;
END_GET
SET
VAR
	button : UINT;
END_VAR
FOR button := 0 TO _config.MaxControlButtons DO
	IF _controlButtons[button] <> 0 THEN
		_controlButtons[button].ButtonRecover := AnyButtonRecover;
	ELSE
		EXIT;
	END_IF
END_FOR
END_SET
END_PROPERTY

{attribute 'monitoring' := 'variable'}
PROPERTY AnyButtonSuspend : BOOL
GET
AnyButtonSuspend := _status.State.AnyButtonSuspend;
END_GET
SET
VAR
	button : UINT;
END_VAR
FOR button := 0 TO _config.MaxControlButtons DO
	IF _controlButtons[button] <> 0 THEN
		_controlButtons[button].ButtonSuspend := AnyButtonSuspend;
	ELSE
		EXIT;
	END_IF
END_FOR
END_SET
END_PROPERTY

METHOD ButtonAuto : BOOL
VAR
	cu : UINT;
END_VAR


IF _autoTask.Execute() THEN
	AnyButtonGround:=FALSE;
	AnyButtonAuto:=_blinkerSlow.IsOn ;		

	IF _autoTask.Progress =0 THEN
	
		IF 	_status.State.AllKeysAuto AND _status.State.AllKeysNormal  THEN
	
			_status.ActionDescription:= '<#Automat mode has been invoked.#>';
			FOR cu := 0 TO _config.MaxControledUnits DO
				IF _controlledUnits[cu] <> 0 THEN
					IF   _controlledUnits[cu].StatusInfo.Mode = eCUMode.GroundModeDone    THEN
						_controlledUnits[cu].AutomatTask.Task.Invoke();
					END_IF	
	
					IF _controlledUnits[cu].StatusInfo.Mode=eCUMode.AutomatMode THEN
							_controlledUnits[cu].AutomatTask.ModeController.Mode:=eSequencerMode.CyclicMode;	
					End_if;	
				ELSE
					EXIT;
				END_IF
			END_FOR
			_autoTask.Progress := _autoTask.Progress + 1;	
			RETURN;
		ELSE
			_status.ActionDescription:= '<#Mode keys are not in correct position.#>';
		END_IF;
			
	ELSE
		
		_autoTask.DoneWhen(_status.State.AllInAuto AND NOT _status.State.AnyButtonAuto);	
		 IF _autoTask.Done THEN
			 
		 	_status.ActionDescription:= '<#Automat mode has been done.#>';
			AnyButtonAuto:=TRUE;
		END_IF;	
	END_IF;
	
	IF _status.ActionDescription<>'' THEN
		THIS^._autoTask.Messenger.Notify(_status.ActionDescription);
	END_IF;
END_IF;
END_METHOD

METHOD ButtonGround : BOOL
VAR
	cu : UINT;
END_VAR

IF _groundTask.Execute() THEN
	// led signalisation
	AnyButtonAuto:=FALSE;
	AnyButtonGround:=_blinkerSlow.IsOn ;	

	IF _groundTask.Progress =0 THEN
		IF 	_status.State.AllKeysAuto AND _status.State.AllKeysNormal  THEN
	
			_status.ActionDescription:= '<#Grounding mode has been invoked.#>';
			FOR cu := 0 TO _config.MaxControledUnits DO
				IF _controlledUnits[cu] <> 0 THEN
					IF  _controlledUnits[cu].StatusInfo.Mode<> eCUMode.GroundMode OR _controlledUnits[cu].StatusInfo.Mode<> eCUMode.GroundModeDone THEN
						_controlledUnits[cu].GroundTask.Task.Invoke();
					END_IF	
					IF _controlledUnits[cu].StatusInfo.Mode=eCUMode.GroundMode THEN
							_controlledUnits[cu].GroundTask.ModeController.Mode:=eSequencerMode.CyclicMode;	
					End_if;			
				ELSE
					EXIT;
				END_IF
			END_FOR
			
			_groundTask.Progress := _groundTask.Progress + 1;	
			RETURN;
		ELSE
			_status.ActionDescription:= '<#Mode keys are not in correct position.#>';
		END_IF;
		
	ELSE
		
		_groundTask.DoneWhen(_status.State.AllGrounded AND NOT _status.State.AnyButtonGround );	
		 IF _groundTask.Done THEN
			 _status.ActionDescription:= '<#Grounding mode has been done.#>';
			AnyButtonGround:=TRUE;
		END_IF;	
	END_IF	
	IF _status.ActionDescription<>'' THEN
		THIS^._groundTask.Messenger.Notify(_status.ActionDescription);
	END_IF;
	

END_IF;
END_METHOD

METHOD ButtonRecover : BOOL
VAR
	cu : UINT;
END_VAR

IF _recoverTask.Execute() THEN
    AnyButtonSuspend := FALSE;

    IF _recoverTask.Progress = 2 THEN
        AnyButtonRecover := _blinker.IsOn;
    ELSE
        AnyButtonRecover := _blinkerSlow.IsOn;
    END_IF;

    IF _recoverTask.Progress = 0 THEN
        FOR cu := 0 TO _config.MaxControledUnits DO
            IF _controlledUnits[cu] <> 0 THEN
                _controlledUnits[cu].RecoverTask.Restore();
            ELSE
                EXIT;
            END_IF
        END_FOR

        _status.ActionDescription := '<#Waiting to release recover button#>';
        IF NOT _status.State.AnyButtonRecover THEN
            _recoverTask.Progress := _recoverTask.Progress + 1;
            RETURN;
        END_IF;

    END_IF

    IF _recoverTask.Progress = 1 THEN
        _status.ActionDescription := '<#Check general condition to recover zone (ControlVoltage, EStops, Presure...)!#>';

        IF inDoorCircuit.IsGlobalVoltageOk AND inDoorCircuit.IsLocalVoltageOk AND inAirPressureOK
        //			AND NOT inEstopActive 
            THEN
            _recoverTask.Progress := _recoverTask.Progress + 1;

        END_IF;

    END_IF

    IF _recoverTask.Progress = 2 THEN
        _status.ActionDescription := '<#Waiting to close and lock  all doors!#>';

        THIS^.inDoorCircuit.Lock();

        IF inDoorCircuit.IsLocked AND inDoorCircuit.IsLocked AND inDoorCircuit.IsLocalDoorsVoltageOk THEN
            _recoverTask.Progress := _recoverTask.Progress + 1;

        END_IF;

    END_IF

    IF _recoverTask.Progress = 3 THEN

        _status.ActionDescription := '<#Invoke restore sequences on each stations.#>';

        IF _status.State.AllInManual OR _status.State.AllInactiveOrManualOrGrounded THEN
            _recoverTask.Progress := 100;
            RETURN;
        END_IF

        FOR cu := 0 TO _config.MaxControledUnits DO
            IF _controlledUnits[cu] <> 0 THEN
                _controlledUnits[cu].RecoverTask.ModeController.Mode := eSequencerMode.CyclicMode;
                _controlledUnits[cu].RecoverTask.Task.Invoke();

            ELSE
                EXIT;
            END_IF
        END_FOR

        IF _status.State.AllRecovered THEN
            _recoverTask.Progress := _recoverTask.Progress + 1;
        END_IF

    END_IF

    IF _recoverTask.Progress = 4 THEN

        _status.ActionDescription := '<#Setup Cyclic or Step mode. It depends on key position#>';

        FOR cu := 0 TO _config.MaxControledUnits DO
            IF _controlledUnits[cu] <> 0 THEN
                IF _status.State.AllKeysAuto THEN
                    IF _controlledUnits[cu].StatusInfo.Mode = eCUMode.AutomatMode THEN
                        _controlledUnits[cu].AutomatTask.ModeController.Mode := eSequencerMode.CyclicMode;
                    ELSIF _controlledUnits[cu].StatusInfo.Mode = eCUMode.GroundMode THEN
                        _controlledUnits[cu].GroundTask.ModeController.Mode := eSequencerMode.CyclicMode;
                    END_IF
                ELSE
                    IF _controlledUnits[cu].StatusInfo.Mode = eCUMode.AutomatMode THEN
                        _controlledUnits[cu].AutomatTask.ModeController.Mode := eSequencerMode.StepMode;
                    ELSIF _controlledUnits[cu].StatusInfo.Mode = eCUMode.GroundMode THEN
                        _controlledUnits[cu].GroundTask.ModeController.Mode := eSequencerMode.StepMode;
                    END_IF
                END_IF

            ELSE
                EXIT;
            END_IF
        END_FOR

        _recoverTask.Progress := 100;

    END_IF

    IF _recoverTask.Progress = 100 THEN

        _status.ActionDescription := '<#Recover task has been done.#>';
        _recoverTask.DoneWhen(TRUE);
        AnyButtonRecover := TRUE;

    END_IF;

    IF _status.ActionDescription <> '' THEN
        THIS^._recoverTask.Messenger.Notify(_status.ActionDescription);
    END_IF;

END_IF;
END_METHOD

METHOD ButtonSuspend : BOOL
VAR
	cu : UINT;
END_VAR
IF _suspendTask.Execute() THEN
	AnyButtonRecover:=FALSE;
	AnyButtonSuspend:=_blinkerSlow.IsOn ;	
	IF _suspendTask.Progress =0 THEN
		FOR cu := 0 TO _config.MaxControledUnits DO
			IF _controlledUnits[cu] <> 0 THEN
				_controlledUnits[cu].SuspendTask.Restore();

			ELSE
				EXIT;
			END_IF
		END_FOR
		_status.ActionDescription:='<#Waiting to release suspend button#>';
		IF NOT _status.State.AnyButtonSuspend THEN
				_suspendTask.Progress := _suspendTask.Progress + 1;	
				RETURN;

		END_IF;
	
	END_IF
	
	IF _suspendTask.Progress =1 THEN
		_status.ActionDescription:='<#Check general condition to suspned zone (ControlVoltage,EStops,Presure...)!#>';
		
		IF NOT inDoorCircuit.IsGlobalVoltageOk
			OR NOT inDoorCircuit.IsLocalVoltageOk
			OR NOT inAirPressureOK
//			OR inEstopActive 
			THEN
			_suspendTask.Progress := 100;
			
			THIS^.inDoorCircuit.Unlock();
		ELSE
			_suspendTask.Progress := _suspendTask.Progress + 1;	
		END_IF;
	
	END_IF
	
	IF _suspendTask.Progress =2 THEN
		
		_status.ActionDescription:= '<#Force step mode.#>';
		
		IF _status.State.AllInManual OR _status.State.AllInactiveOrManualOrGrounded THEN
			_suspendTask.Progress := 4;
			RETURN;
		END_IF
		FOR cu := 0 TO _config.MaxControledUnits DO
			IF _controlledUnits[cu] <> 0 THEN
			

				IF _controlledUnits[cu].StatusInfo.Mode=eCUMode.AutomatMode THEN
					_controlledUnits[cu].AutomatTask.ModeController.Mode:=eSequencerMode.StepMode;
				ELSIF _controlledUnits[cu].StatusInfo.Mode=eCUMode.GroundMode THEN
					_controlledUnits[cu].GroundTask.ModeController.Mode:=eSequencerMode.StepMode;
				END_IF
		
	
			ELSE
				EXIT;
			END_IF
		END_FOR


		
		IF _status.State.AllInStepMode or true THEN
			_suspendTask.Progress := _suspendTask.Progress + 1;
		END_IF;
			
	END_IF
	
	IF _suspendTask.Progress =3 THEN
		
		_status.ActionDescription:='<#Invoke suspend sequences on each stations.#>';
		
		
		FOR cu := 0 TO _config.MaxControledUnits DO
			IF _controlledUnits[cu] <> 0 THEN
				_controlledUnits[cu].SuspendTask.ModeController.Mode := eSequencerMode.CyclicMode;
				_controlledUnits[cu].SuspendTask.Task.Invoke();

			ELSE
				EXIT;
			END_IF
		END_FOR

		IF _status.State.AllSuspended THEN
			_suspendTask.Progress := _suspendTask.Progress+1;
		END_IF
		
	END_IF
	
	
	
	IF _suspendTask.Progress =4 THEN
		_status.ActionDescription:='<#Waiting to unlock  all doors!#>';
		
		THIS^.inDoorCircuit.UnLock();
		
		IF inDoorCircuit.IsUnLocked THEN
		//	_suspendTask.Progress := 100;
	
		END_IF;
	
	END_IF


	IF _suspendTask.Progress = 100 THEN
		_status.ActionDescription:= '<#Suspend task has been done.#>';
		_suspendTask.DoneWhen(TRUE);
		AnyButtonSuspend:=TRUE;
	END_IF;	


	IF _status.ActionDescription<>'' THEN
		THIS^._suspendTask.Messenger.Notify(_status.ActionDescription);
	END_IF;
	
END_IF;
END_METHOD

PROPERTY Config :REFERENCE TO TcoControlledZone_Config
GET
Config ref=_config;
END_GET
END_PROPERTY

METHOD Initialize : BOOL
VAR
	i : UINT;

END_VAR
_status.State.AllInAuto := TRUE;
_status.State.AllInGrounding := TRUE;
_status.State.AllInManual := TRUE;
_status.State.AllIdle := TRUE;
_status.State.AllGrounded := TRUE;
_status.State.AllInStepMode := TRUE;
_status.State.AllSuspended := TRUE;
_status.State.AllRecovered := TRUE;
_status.State.AllInactiveOrManualOrGrounded :=true;
_status.State.AnyInAuto := FALSE;
_status.State.AnyInManual := FALSE;
_status.State.AnyGrounding := FALSE;
_status.State.AnyInStepMode := FALSE;

i := 0;

FOR i := 0 TO _config.MaxControledUnits DO
    IF _controlledUnits[i] <> 0 THEN
        _status.State.AllInAuto := _status.State.AllInAuto AND _controlledUnits[i].StatusInfo.Mode = eCUMode.AutomatMode;
        _status.State.AllInManual := _status.State.AllInManual AND _controlledUnits[i].StatusInfo.Mode = eCUMode.ManualMode;
        _status.State.AllIdle := _status.State.AllIdle AND _controlledUnits[i].StatusInfo.Mode = eCUMode.NoMode;
        _status.State.AllInGrounding := _status.State.AllInGrounding AND
            (_controlledUnits[i].StatusInfo.Mode = eCUMode.GroundModeDone XOR
            _controlledUnits[i].StatusInfo.Mode = eCUMode.GroundMode);
        _status.State.AllGrounded := _status.State.AllGrounded AND _controlledUnits[i].StatusInfo.Mode = eCUMode.GroundModeDone;
        _status.State.AllInStepMode := _status.State.AllInStepMode AND _controlledUnits[i].StatusInfo.CurrentIsInStepMode;
        _status.State.AllSuspended := _status.State.AllSuspended AND _controlledUnits[i].SuspendTask.Task.Done;
		_status.State.AllRecovered := _status.State.AllRecovered AND _controlledUnits[i].RecoverTask.Task.Done;
		_status.State.AllInactiveOrManualOrGrounded := _status.State.AllInactiveOrManualOrGrounded 
											AND (_controlledUnits[i].StatusInfo.Mode = eCUMode.ManualMode 
												OR _controlledUnits[i].StatusInfo.Mode = eCUMode.NoMode 
												OR _controlledUnits[i].StatusInfo.Mode = eCUMode.GroundModeDone );
		
        _status.State.AnyInAuto := _status.State.AnyInAuto OR _controlledUnits[i].StatusInfo.Mode = eCUMode.AutomatMode;
        _status.State.AnyInManual := _status.State.AnyInManual OR _controlledUnits[i].StatusInfo.Mode = eCUMode.ManualMode;
        _status.State.AnyInStepMode := _status.State.AnyInStepMode OR _controlledUnits[i].StatusInfo.CurrentIsInStepMode;
        _status.State.AnyGrounding := _status.State.AnyGrounding OR
            (_controlledUnits[i].StatusInfo.Mode = eCUMode.GroundModeDone OR
            _controlledUnits[i].StatusInfo.Mode = eCUMode.GroundMode);

    ELSE
        EXIT;
    END_IF
END_FOR

// update states of buttons
_status.State.AnyButtonRecover := FALSE;
_status.State.AnyButtonSuspend := FALSE;
_status.State.AnyButtonGround := FALSE;
_status.State.AnyButtonAuto := FALSE;
i := 0;

FOR i := 0 TO _config.MaxControlButtons DO
    IF _controlButtons[i] <> 0 THEN
        _status.State.AnyButtonRecover := _status.State.AnyButtonRecover OR _controlButtons[i].ButtonRecover;
        _status.State.AnyButtonGround := _status.State.AnyButtonGround OR _controlButtons[i].ButtonGround;
        _status.State.AnyButtonAuto := _status.State.AnyButtonAuto OR _controlButtons[i].ButtonAuto;
        _status.State.AnyButtonSuspend := _status.State.AnyButtonSuspend OR _controlButtons[i].ButtonSuspend;
    ELSE
        EXIT;
    END_IF
END_FOR

// update states of keys
_status.State.AllKeysNormal := TRUE;
_status.State.AnyKeyService := FALSE;
i := 0;

FOR i := 0 TO _config.MaxKeyNormalService DO
    IF _controlKeyNormalService[i] <> 0 THEN
        _status.State.AllKeysNormal := _status.State.AllKeysNormal AND _controlKeyNormalService[i].KeyInNormal;
        _status.State.AnyKeyService := _status.State.AnyKeyService OR _controlKeyNormalService[i].KeyInService;
    ELSE
        EXIT;
    END_IF
END_FOR

// update states of keys
_status.State.AllKeysAuto := TRUE;
_status.State.AnyKeyManual := FALSE;
_status.State.AnyKeyStep := FALSE;
i := 0;

FOR i := 0 TO _config.MaxKeyMode DO
    IF _controlKeyMode[i] <> 0 THEN
        _status.State.AllKeysAuto := _status.State.AllKeysAuto AND _controlKeyMode[i].KeyInAuto;
        _status.State.AnyKeyManual := _status.State.AnyKeyManual OR _controlKeyMode[i].KeyInManual;
        _status.State.AnyKeyStep := _status.State.AnyKeyStep OR _controlKeyMode[i].KeyInStep;
    ELSE
        EXIT;
    END_IF
END_FOR
END_METHOD

METHOD KeyAuto 
VAR
	cu : UINT;
END_VAR
IF _keyAutoTask.Execute() THEN
	_status.ActionDescription:= '<#Automatic mode is not possibe to set(All keys must be in NORMAL and AUTO!)#>';
	IF 	 _status.State.AllKeysNormal  AND _status.State.AllKeysAuto THEN
		
//			_status.ActionDescription:= '<#Automatic mode is set(Step mode is disabled)!#>';
//			FOR cu := 0 TO _config.MaxControledUnits DO
//				IF _controlledUnits[cu] <> 0 THEN
//					IF _controlledUnits[cu].StatusInfo.Mode=eCUMode.AutomatMode THEN
//						_controlledUnits[cu].AutomatTask.ModeController.Mode:=eSequencerMode.CyclicMode;
//					ELSIF _controlledUnits[cu].StatusInfo.Mode=eCUMode.GroundMode THEN
//						_controlledUnits[cu].GroundTask.ModeController.Mode:=eSequencerMode.CyclicMode;
//					END_IF
//				ELSE
//					EXIT;
//				END_IF
//			END_FOR
	
		ELSE
			_status.ActionDescription:= '<#Cyclic mode is not allowed while any control key is in Service mode!#> <#Setting step mode!#>';
			FOR cu := 0 TO _config.MaxControledUnits DO
				IF _controlledUnits[cu] <> 0 THEN
						IF _controlledUnits[cu].StatusInfo.Mode=eCUMode.AutomatMode THEN
							_controlledUnits[cu].AutomatTask.ModeController.Mode:=eSequencerMode.StepMode;
						ELSIF _controlledUnits[cu].StatusInfo.Mode=eCUMode.GroundMode THEN
							_controlledUnits[cu].GroundTask.ModeController.Mode:=eSequencerMode.StepMode;
						END_IF
				ELSE
					EXIT;
				END_IF
			END_FOR	
		END_IF;
	
	


	IF  _status.State.AllInAuto THEN
		_keyAutoTask.DoneWhen(TRUE);
	END_IF;
	
	IF _status.ActionDescription<>'' THEN
		THIS^._keyAutoTask.Messenger.Notify(_status.ActionDescription);
	END_IF;	
END_IF
END_METHOD

METHOD KeyManual 
VAR
	cu : UINT;
END_VAR

IF _keyManualTask.Execute() THEN
	_status.ActionDescription:= '<#Manual mode is not possibe to set(At least one SERVICE and one MANUAL keys must be in position!)#>';
	
	IF _keyManualTask.Progress =0 THEN
		IF _status.State.AnyKeyManual AND _status.State.AnyKeyService THEN
			IF NOT _status.State.AllInManual THEN
				_keyManualTask.Progress := _keyManualTask.Progress + 1;// all to manual
			ELSE
				_keyManualTask.Progress := _keyManualTask.Progress + 2;
			END_IF
		END_IF;
	
	END_IF

	IF _keyManualTask.Progress =1 THEN
		
		_status.ActionDescription:='<#Manual mode is starting#>';
		
		FOR cu := 0 TO _config.MaxControledUnits DO
			IF _controlledUnits[cu] <> 0 THEN
				IF  _controlledUnits[cu].StatusInfo.Mode<> eCUMode.ManualMode THEN
					_controlledUnits[cu].ManualTask.Invoke();
				END_IF			
			ELSE
				EXIT;
			END_IF
		END_FOR

		IF _status.State.AllInManual THEN
			_keyManualTask.Progress := _keyManualTask.Progress + 1;
		END_IF
		
	END_IF
	
	
	IF _keyManualTask.Progress =2 THEN
		
		_status.ActionDescription:='<#Clear step mode#>';
		
		FOR cu := 0 TO _config.MaxControledUnits DO
			IF _controlledUnits[cu] <> 0 THEN
				_controlledUnits[cu].AutomatTask.ModeController.Mode := eSequencerMode.CyclicMode;
				_controlledUnits[cu].GroundTask.ModeController.Mode := eSequencerMode.CyclicMode;		
			ELSE
				EXIT;
			END_IF
		END_FOR

		IF _status.State.AllInManual THEN
			_keyManualTask.Progress := _keyManualTask.Progress + 1;
		END_IF
		
	END_IF

	IF _keyManualTask.Progress =3 THEN
		_keyManualTask.DoneWhen(TRUE);	
	END_IF

	IF _status.ActionDescription<>'' THEN
		THIS^._keyManualTask.Messenger.Notify(_status.ActionDescription);
	END_IF;
END_IF;
END_METHOD

METHOD KeyService
VAR
	cu : UINT;
END_VAR
IF _keyServiceTask.Execute() THEN
	
	IF 	_status.State.AnyKeyManual  AND _status.State.AnyKeyService  THEN
		_status.ActionDescription:='<#Manual mode is starting due service key combination (Manual / Service)#>';
		
		FOR cu := 0 TO _config.MaxControledUnits DO
			IF _controlledUnits[cu] <> 0 THEN
				IF  _controlledUnits[cu].StatusInfo.Mode<> eCUMode.ManualMode THEN
					_controlledUnits[cu].ManualTask.Invoke();
				END_IF			
			ELSE
				EXIT;
			END_IF
		END_FOR
	ELSE
		_status.ActionDescription:='<#Step mode is required because Service key position is set!#>';
		FOR cu := 0 TO _config.MaxControledUnits DO
			IF _controlledUnits[cu] <> 0 THEN
					IF _controlledUnits[cu].StatusInfo.Mode=eCUMode.AutomatMode THEN
						_controlledUnits[cu].AutomatTask.ModeController.Mode:=eSequencerMode.StepMode;
					ELSIF _controlledUnits[cu].StatusInfo.Mode=eCUMode.GroundMode THEN
						_controlledUnits[cu].GroundTask.ModeController.Mode:=eSequencerMode.StepMode;
					END_IF
			ELSE
				EXIT;
			END_IF
		END_FOR
	END_IF;
	


	IF  _status.State.AllInStepMode OR _status.State.AllInManual THEN
		_keyServiceTask.DoneWhen(TRUE);
	END_IF;
	
	IF _status.ActionDescription<>'' THEN
		THIS^._keyServiceTask.Messenger.Notify(_status.ActionDescription);
	END_IF;	
END_IF
END_METHOD

METHOD KeyStep 
VAR
	cu : UINT;
END_VAR

IF _keyStepTask.Execute() THEN
		
	_status.ActionDescription:='<#Step mode is required but mode key is not in required position!#>';

	IF _status.State.AnyKeyStep THEN
		FOR cu := 0 TO _config.MaxControledUnits DO
			IF _controlledUnits[cu] <> 0 THEN
				IF _controlledUnits[cu].StatusInfo.Mode=eCUMode.AutomatMode THEN
					_controlledUnits[cu].AutomatTask.ModeController.Mode:=eSequencerMode.StepMode;
				ELSIF _controlledUnits[cu].StatusInfo.Mode=eCUMode.GroundMode THEN
					_controlledUnits[cu].GroundTask.ModeController.Mode:=eSequencerMode.StepMode;
				END_IF
			ELSE
				EXIT;
			END_IF
		
		END_FOR
	END_IF;
	
	IF _status.State.AllInStepMode THEN
		_status.ActionDescription:='<#Step mode is set or all are inactive!#>';
		_keyStepTask.DoneWhen(TRUE);
	END_IF;
	
	IF _status.ActionDescription<>'' THEN
		THIS^._keyStepTask.Messenger.Notify(_status.ActionDescription);
	END_IF;	
END_IF;
END_METHOD

METHOD Restore :  TcoCore.ITcoRestorable
VAR
	i : UINT;
END_VAR
// clear all linked Controlled units
FOR i := 0 TO _config.MaxControledUnits DO
	_controlledUnits[i] := 0;
END_FOR

// clear all linked Control buttons
FOR i := 0 TO _config.MaxControlButtons DO
	_controlButtons[i] := 0;
END_FOR

// clear all linked service keys (N/S)
FOR i := 0 TO _config.MaxKeyNormalService DO
	_controlKeyNormalService[i] := 0;
END_FOR

// clear all linked Sequencer keys (M/S/A)
FOR i := 0 TO _config.MaxKeyMode DO
	_controlKeyMode[i] := 0;
END_FOR


THIS^.Messenger.UnPin();
END_METHOD

(*~
	<docu>
		<summary>
		    Custom service (manual, maintenance) logic.
			This method must be implemented in derived class.
		</summary>			
	</docu>	
~*)
METHOD PROTECTED  ServiceMode
END_METHOD

METHOD Signalisation
VAR_INPUT
END_VAR

AnyButtonAuto:=_blinkerSlow.IsOn  AND _autoTask.Busy;
END_METHOD

PROPERTY Status : REFERENCE TO TcoControlledZone_Status
GET
Status REF=_status;
END_GET
END_PROPERTY

END_FUNCTION_BLOCK

// ---- Abstractions/Safety/DoorCircuit/TcoDoorCircuit.TcPOU
FUNCTION_BLOCK TcoDoorCircuit EXTENDS TcoCore.TcoComponent IMPLEMENTS ITcoDoorCircuit
VAR_INPUT
END_VAR
VAR_OUTPUT
END_VAR
VAR
	
	{attribute addProperty Name "<#Status#>"}
    {attribute clr [ReadOnly()]}
    _status : TcoDoorCircuit_Status;

	{attribute addProperty Name "<#Config#>"}
    _config : TcoDoorCircuit_Config;

	
	//~
	_doors              : ARRAY [0..12] OF ITcoDoorLock;
	
	{attribute clr [RenderIgnore()]}
	_localDoorsVoltage  : ARRAY [0..4] OF ITcoControlVoltage;
	
	{attribute clr [RenderIgnore()]}
	_localVoltage  : ARRAY [0..4] OF ITcoControlVoltage;
	
	{attribute clr [RenderIgnore()]}
	_globalVoltage : ARRAY [0..4] OF ITcoControlVoltage;
	//~
	
	
    {attribute addProperty Name "<#Closed#>"}
    _isClosed : BOOL;
    
    {attribute addProperty Name "<#Locked#>"}
    _isLocked : BOOL;
    
    {attribute addProperty Name "<#Unlocked#>"}
    _isUnLocked : BOOL;
    
    {attribute addProperty Name "<#Global votage#>"}
    _isGlobalVoltageOk : BOOL;
    
    {attribute addProperty Name "<#Local voltage#>"}
    _isLocalVoltageOk : BOOL;
    
	 {attribute addProperty Name "<#Local Doors#>"}
    _isLocalDoorsVoltageOk : BOOL;


END_VAR

Initialize();

METHOD AddDoors : BOOL
VAR_INPUT
	inDoor : ITcoDoorLock;
END_VAR
VAR
	i : UINT;
END_VAR
AddDoors := FALSE;
FOR i := 0 TO _config.MaxDoors DO
	IF _doors[i] = inDoor THEN
		AddDoors := TRUE;
		RETURN;
	END_IF
	
	IF _doors[i] = 0 THEN
		_doors[i] := inDoor;
		AddDoors := TRUE;
		RETURN;
	END_IF
END_FOR
END_METHOD

METHOD AddGlobalVoltage : BOOL
VAR_INPUT
 	inVoltage : ITcoControlVoltage;
END_VAR
VAR
	i : UINT;
END_VAR
AddGlobalVoltage := FALSE;

IF inVoltage = 0 THEN
	RETURN;
END_IF

FOR i := 0 TO _config.MaxGlobalVoltage DO
	IF _globalVoltage[i] = inVoltage THEN
		addGlobalVoltage := TRUE;
		RETURN;
	END_IF
	
	IF 	_globalVoltage[i] = 0 THEN
		_globalVoltage[i] := inVoltage;
		addGlobalVoltage    := TRUE;
		RETURN;
	END_IF
END_FOR
END_METHOD

METHOD AddLocalDoorsVoltage : BOOL
VAR_INPUT
 	inVoltage : ITcoControlVoltage;
END_VAR
VAR
	i : UINT;
END_VAR
AddLocalDoorsVoltage := FALSE;

IF inVoltage = 0 THEN
	RETURN;
END_IF

FOR i := 0 TO _config.MaxLocalVoltage DO
	IF _localDoorsVoltage[i] = inVoltage THEN
		AddLocalDoorsVoltage := TRUE;
		RETURN;
	END_IF
	
	IF 	_localDoorsVoltage[i] = 0 THEN
		_localDoorsVoltage[i] := inVoltage;
		AddLocalDoorsVoltage    := TRUE;
		RETURN;
	END_IF
END_FOR
END_METHOD

METHOD AddLocalVoltage : BOOL
VAR_INPUT
 	inVoltage : ITcoControlVoltage;
END_VAR
VAR
	i : UINT;
END_VAR
addLocalVoltage := FALSE;

IF inVoltage = 0 THEN
	RETURN;
END_IF

FOR i := 0 TO _config.MaxLocalVoltage DO
	IF _localVoltage[i] = inVoltage THEN
		addLocalVoltage := TRUE;
		RETURN;
	END_IF
	
	IF 	_localVoltage[i] = 0 THEN
		_localVoltage[i] := inVoltage;
		addLocalVoltage    := TRUE;
		RETURN;
	END_IF
END_FOR
END_METHOD

PROPERTY Config :REFERENCE TO TcoDoorCircuit_Config
GET
Config ref=_config;
END_GET
END_PROPERTY

METHOD Initialize : BOOL
VAR
	d       : UINT;
	gv      : UINT;
	lv      : UINT;
	ldoors      : UINT;
	setOnce : BOOL;
END_VAR
// ------------------------------------------------------------- 
// 						GLOBAL VOLTAGE
// ------------------------------------------------------------- 
_isGlobalVoltageOk := FALSE;
setOnce            := FALSE;

FOR gv := 0 TO _config.MaxGlobalVoltage DO
	IF _globalVoltage[gv] <> 0 THEN
		IF NOT setOnce THEN
			_isGlobalVoltageOk := TRUE;
			setOnce := TRUE;
		END_IF
		
		IF _globalVoltage[gv].IsOff THEN
			_isGlobalVoltageOk := FALSE;
			EXIT;
		END_IF
	ELSE
		EXIT;
	END_IF
END_FOR

// ------------------------------------------------------------- 
// 						LOCAL VOLTAGE
// ------------------------------------------------------------- 
_isLocalVoltageOk := FALSE;
setOnce           := FALSE;

FOR lv := 0 TO _config.MaxLocalVoltage DO
	IF _localVoltage[lv] <> 0 THEN
		IF NOT setOnce THEN
			_isLocalVoltageOk := TRUE;
			setOnce := TRUE;
		END_IF
		
		IF _localVoltage[lv].IsOff THEN
			_isLocalVoltageOk := false;
			EXIT;
		END_IF
	ELSE
		EXIT;
	END_IF
END_FOR

// ------------------------------------------------------------- 
// 						LOCAL DOORS VOLTAGE OK
// ------------------------------------------------------------- 
_isLocalDoorsVoltageOk := FALSE;
setOnce           := FALSE;

FOR ldoors := 0 TO _config.MaxLocalDoorsVoltage DO
	IF _localDoorsVoltage[ldoors] <> 0 THEN
		IF NOT setOnce THEN
			_isLocalDoorsVoltageOk := TRUE;
			setOnce := TRUE;
		END_IF
		
		IF _localDoorsVoltage[ldoors].IsOff THEN
			_isLocalDoorsVoltageOk := FALSE;
			EXIT;
		END_IF
	ELSE
		EXIT;
	END_IF
END_FOR

// ------------------------------------------------------------- 
// 							DOORS
// ------------------------------------------------------------- 
_isClosed      := FALSE;
_isLocked      := FALSE;
_isUnLocked    := FALSE;
setOnce        := FALSE;
FOR d := 0 TO _config.MaxDoors DO
	IF _doors[d] <> 0 THEN
		IF NOT setOnce THEN
			setOnce        := TRUE;
			_isClosed      := TRUE;
			_isLocked      := TRUE;
			_isUnLocked    := TRUE;
		END_IF

		// Return TRUE only if all doors are Closed
		_isClosed   := _isClosed AND (_doors[d].IsClosed); // OR _doors[d].Deactivate);
		// Return TRUE only if all doors are Locked
		_isLocked   := _isLocked AND (_doors[d].IsLocked); //OR _doors[d].Deactivate);
		// Return TRUE only if all doors are Unlocked
		_isUnLocked := _isUnLocked AND NOT _doors[d].IsLocked;

	ELSE
		EXIT;
	END_IF
END_FOR
END_METHOD

{attribute 'monitoring' := 'variable'}
PROPERTY IsClosed : BOOL
GET
VAR
	d : UINT;
	setOnce : BOOL;
END_VAR
IsClosed := _isClosed ;
END_GET
END_PROPERTY

{attribute 'monitoring' := 'variable'}
PROPERTY IsGlobalVoltageOk : BOOL
GET
VAR
	gv : UINT;
END_VAR
IsGlobalVoltageOk := _isGlobalVoltageOk;
END_GET
END_PROPERTY

{attribute 'monitoring' := 'variable'}
PROPERTY IsLocalDoorsVoltageOk : BOOL
GET
VAR
	lv : UINT;
END_VAR
IsLocalDoorsVoltageOk := _isLocalDoorsVoltageOk;
END_GET
END_PROPERTY

{attribute 'monitoring' := 'variable'}
PROPERTY IsLocalVoltageOk : BOOL
GET
VAR
	lv : UINT;
END_VAR
IsLocalVoltageOk := _isLocalVoltageOk;
END_GET
END_PROPERTY

{attribute 'monitoring' := 'variable'}
PROPERTY IsLocked : BOOL
GET
VAR
	d : UINT;
	setOnce : BOOL;
END_VAR
IsLocked := _isLocked ;
END_GET
END_PROPERTY

{attribute 'monitoring' := 'variable'}
PROPERTY IsUnLocked : BOOL
GET
VAR
	d : UINT;
	setOnce : BOOL;
END_VAR
IsUnLocked := _isUnLocked;
END_GET
END_PROPERTY

METHOD Lock : BOOL
VAR_INPUT
END_VAR
VAR
	d : UINT;
END_VAR
Lock := FALSE;

IF NOT IsClosed THEN
	// we can't lock doors which are not closed
	RETURN;
END_IF

FOR d := 0 TO _config.MaxDoors DO
	IF _doors[d] <> 0 THEN
			_doors[d].Lock();
	ELSE
		EXIT;
	END_IF
END_FOR

Lock := THIS^.IsLocked;
END_METHOD

METHOD RemoveAllDoors
VAR
	i : UINT;
END_VAR
FOR i := 0 TO _config.MaxDoors DO
	_doors[i] := 0;
END_FOR
END_METHOD

METHOD RemoveDoors : BOOL
VAR_INPUT
	inDoorLock : ITcoDoorLock;
END_VAR
VAR
	i : UINT;
END_VAR
RemoveDoors := FALSE;

FOR i := 0 TO _config.MaxDoors DO 
	IF _doors[i] = inDoorLock THEN
		_doors[i] := 0;
		RemoveDoors :=  TRUE;
		RETURN;
	END_IF
END_FOR
END_METHOD

(*~
	<docu>
		<summary>
			Restores this instance to the Ready state. Can be called explicitly or from within one of the restore mechanisms.	
		</summary>			
	</docu>	
~*)
METHOD  Restore : ITcoRestorable

VAR
	i : UINT;
END_VAR
RemoveAllDoors();

FOR i := 0 TO _config.MaxGlobalVoltage DO
	_globalVoltage[i] := 0;
END_FOR

FOR i := 0 TO _config.MaxLocalVoltage DO
	_localVoltage[i] := 0;
END_FOR
FOR i := 0 TO _config.MaxLocalDoorsVoltage DO
	_localDoorsVoltage[i] := 0;
END_FOR
END_METHOD

(*~
	<docu>
		<summary>
		    Custom service (manual, maintenance) logic.
			This method must be implemented in derived class.
		</summary>			
	</docu>	
~*)
METHOD PROTECTED  ServiceMode
END_METHOD

PROPERTY Status : REFERENCE TO TcoDoorCircuit_Status
GET
Status REF=_status;
END_GET
END_PROPERTY

METHOD UnLock : BOOL
VAR
	d 		: UINT;
	setOnce : BOOL;
END_VAR
UnLock := FALSE;

FOR d := 0 TO _config.MaxDoors DO
	IF _doors[d] <> 0 THEN
		_doors[d].Unlock();
	ELSE
		exit;
	END_IF
END_FOR


FOR d := 0 TO _config.MaxDoors DO
	IF _doors[d] <> 0 THEN
		IF NOT setOnce THEN
			setOnce := TRUE;
			UnLock := TRUE;
		END_IF
		
		// return TRUE only if all doors are unlocked
		UnLock := Unlock AND NOT _doors[d].IsLocked;
	ELSE
		EXIT;
	END_IF
END_FOR
END_METHOD

END_FUNCTION_BLOCK

// ---- Technology/CU00x/Automat/CU00xAutomatParalell_1_Task.TcPOU
FUNCTION_BLOCK CU00xAutomatParalell_1_Task EXTENDS TcoTaskedSequencer 

VAR
	_customTimer: TON;
END_VAR

Run();

(*~
	<docu>
		<summary>
			Main method of the sequener. Custom code needs to be placed here. The sequencer is executed by call of **Instance.Run()** method.
			This method is abstract, and it must be overridden in derived block.
		</summary>
	</docu>
~*)
METHOD PROTECTED Main : BOOL
// Takes mode (step/continous) from the parent controller
THIS^.ModeController.Mode := ParentSequence.ModeController.Mode;

IF (Step(1000, TRUE, 'PARALELL STEP - EXAMPLE OF TIMERS')) THEN
    //-------------------------------------    
		StepCompleteWhen(CurrentStep.Duration >= T#300mS);	
    //-------------------------------------
END_IF
IF (Step(1100, TRUE, 'PARALELL STEP - EXAMPLE OF TIMERS')) THEN
    //-------------------------------------    
		StepCompleteWhen(inCondition:=Timer_1(TRUE,T#100MS));	
    //-------------------------------------
END_IF
IF (Step(1200, TRUE, 'PARALELL STEP - EXAMPLE OF TIMERS')) THEN
    //-------------------------------------    
		StepCompleteWhen(inCondition:=Timer_1(TRUE,T#200MS));	
    //-------------------------------------
END_IF


IF THIS^.IsFreshState THEN
	_customTimer(IN:=FALSE);
END_IF
IF (Step(1300, TRUE, 'PARALELL STEP - EXAMPLE OF TIMERS')) THEN
    //-------------------------------------    

		_customTimer(IN:=TRUE,PT:=T#200MS);
		StepCompleteWhen(inCondition:=_customTimer.Q);	
    //-------------------------------------
END_IF


IF (Step(10000, TRUE, 'PARALELL TASK DONE')) THEN
    //-------------------------------------
    _task.DoneWhen(TRUE );
    //-------------------------------------	
END_IF
END_METHOD

PROPERTY ParentSequence : REFERENCE TO CU00xAutomatTask
GET
VAR
    _parentSequence : POINTER TO CU00xAutomatTask;
END_VAR
IF __QUERYPOINTER(Parent, _parentSequence) THEN 
    ParentSequence REF= _parentSequence^;              
END_IF
END_GET
END_PROPERTY

END_FUNCTION_BLOCK

// ---- Technology/CU00x/Automat/CU00xAutomatTask.TcPOU
FUNCTION_BLOCK CU00xAutomatTask EXTENDS CUBaseAutomat IMPLEMENTS ICUTask
VAR

    _missingProcessSettingMessage : TcoCore.TcoMessenger(THIS^);
    _paralellTask : CU00xAutomatParalell_1_Task(THIS^, TcoCore.eRestoreMode.None);
	
	//~
    _sb : TcoCore.StringBuilder;
	//~
    _customizedContentInput : CU00xDialogContent(THIS^);
END_VAR

VAR
    _dataLoadProcessSettings : BOOL;
    _dataLoadProcessSettingsByPlaner : BOOL;
    _dataCreateNew : BOOL;
    _dataOpen : BOOL;
    _dataClose : BOOL;
    _dataFinalize : BOOL;
    _continueRestore : BOOL;
    _loop : BOOL;
    _inspectionResult : BOOL;
    _inspectionDimensionResult : REAL;
    _tagsPairing : BOOL;
    _reqKey : STRING;
    _reqAssignedValue : STRING;
    _inspectorSingleExamples : BOOL;
    _inspectorGroupExamples : BOOL;
	_dialogExamples : BOOL;

END_VAR

Run();

(*~
	<docu>
		<summary>
			Loads technology settings from the current technology set into this controlled unit.
			The `StationProcessDataManager.Data` is populated by data from process settings.						
		</summary>
	</docu>
~*)
METHOD DataLoadProcessSettings : BOOL
VAR_INPUT
	inStepID : INT;
END_VAR

VAR
	_ans: TcoCore.eDialogAnswer;
END_VAR
IF (Step(inStepID, _dataLoadProcessSettings, 'LOAD PROCESS SETTING')) THEN
    //-------------------------------------
	
	THIS^._missingProcessSettingMessage.OnCondition(Station.Technology.ProcessSettings.Data._EntityId = '')
									   .Build()
									   .Append('No process data. Please load setting')
									   .As()				   
									   .AsError()
									   .Pin();
					   
				   
	IF(Station.Technology.ProcessSettings.Data._EntityId <> '' (*AND NOT THIS^._missingProcessSettingMessage.Pinned*)) THEN
		IF(Station.Technology.ProcessSettings.Read(Station.Technology.ProcessSettings.Data._EntityId).Done) THEN
			Station.ProcessDataManager.Data := Station.Technology.ProcessSettings.Data;
			Station.ProcessDataManager.Data.EntityHeader.RecipeCreated := Station.Technology.ProcessSettings.Data._Created;
			Station.ProcessDataManager.Data.EntityHeader.RecipeLastModified  := Station.Technology.ProcessSettings.Data._Modified;
			Station.ProcessDataManager.Data.EntityHeader.Recipe  := Station.Technology.ProcessSettings.Data._EntityId;				
			CompleteStep();

		END_IF;	
	ELSE
		_ans:=_dialog.Show()
			.WithImage('d:\MTS\Develop\TcOpenGroup\TcOpen\assets\logo\TcOpenWide.png',400,600)	
	       .WithCaption('<#Process data not selected#>')
		   .WithText('<#Would you like to load default settings?#>')
		   .WithYesNoCancel().Answer;
		IF(_ans=TcoCore.eDialogAnswer.Cancel) THEN
			this^.Restore();
		END_IF
		IF( _ans= TcoCore.eDialogAnswer.Yes) THEN
		   
		   	Station.Technology.ProcessSettings.Data._EntityId := 'default';
		END_IF; 

			
	END_IF		    				
    //-------------------------------------
END_IF
END_METHOD

(*~
	<docu>
		<summary>
			Loads process settings from the current process set into this controlled unit.
			The `StationProcessDataManager.Data` is populated by data from process settings.						
		</summary>
	</docu>
~*)
METHOD DataLoadProcessSettingsByPlaner : BOOL
VAR_INPUT
	inStepID : INT;
END_VAR
IF (Step(inStepID, _dataLoadProcessSettingsByPlaner, 'LOAD PROCESS SETTING BY THE PRODUCTION PLANER')) THEN
    //-------------------------------------


								   
	 IF Station.ProductionPlanerTask.Invoke().Done	AND_THEN(Station.ProductionPlanerTask.RequiredProcessSettingsId <> '') THEN
		
		IF NOT Station.ProductionPlanerTask.ProductionPlanCompleted and_then (Station.Technology.ProcessSettings.Read(Station.ProductionPlanerTask.RequiredProcessSettingsId).Done)
			 THEN
			Station.ProcessDataManager.Data := Station.Technology.ProcessSettings.Data;
			Station.ProcessDataManager.Data.EntityHeader.RecipeCreated := Station.Technology.ProcessSettings.Data._Created;
			Station.ProcessDataManager.Data.EntityHeader.RecipeLastModified  := Station.Technology.ProcessSettings.Data._Modified;
			Station.ProcessDataManager.Data.EntityHeader.Recipe  := Station.Technology.ProcessSettings.Data._EntityId;				
			CompleteStep();
			Station.ProductionPlanerTask.Restore();
		END_IF;
	ELSIF  Station.ProductionPlanerTask.ProductionPlanIsEmpty THEN
		IF (_dialog.Show()
	       .WithCaption('<#Production planer#>')
		   .WithText('<#Production planer is empty!#>')
			.WithOk().Answer = TcoCore.eDialogAnswer.OK) THEN;
			;// Production plan comleted , here you can write diferent scenario ( leave it with current state , provide ground etc)	 
	
		 	//Station.GroundTask.Task.Invoke();
		   
		End_if;
	
	ELSIF  Station.ProductionPlanerTask.ProductionPlanCompleted THEN
		IF (_dialog.Show()
	       .WithCaption('<#Production planer#>')
		   .WithText('<#Production planer completed required plan!#>')
			.WithOk().Answer = TcoCore.eDialogAnswer.OK) THEN;
			;// Production plan comleted , here you can write diferent scenario ( leave it with current state , provide ground etc)	 
	
		 	//Station.GroundTask.Task.Invoke();
		   
		End_if;

			
	END_IF		    				
    //-------------------------------------
END_IF
END_METHOD

(*~
	<docu>
		<summary>
			Wait for start operations and then go into this controlled unit sequence.						
		</summary>
	</docu>
~*)
METHOD DataReadyForOperations : BOOL
VAR_INPUT
	inStepID : INT;
END_VAR

VAR
	_ans: TcoCore.eDialogAnswer;
END_VAR
THIS^.Station.ResetReadyForOperations();   

IF (Step(inStepID, TRUE, '<#READY TO START OPERATIONS#>')) THEN
    //-------------------------------------
	
	THIS^.Station.SetReadyForOperations();   
	
  	Await(THIS^.Station.InternalRetrieveEntity(inCarrier:=2(*here comes info from carousel position*),refStorage:=Station.Technology.InternalStorage) 
			 AND_THEN THIS^.Station.DoesBelong() 
			 AND_THEN THIS^.Station.RunOperations(refGlobalTrigger:=Station.Technology.RunOperations)
			 AND_THEN THIS^.Station.InternalOpenEntity(inCarrier:=2(*here comes info from carousel position*),refStorage:=Station.Technology.InternalStorage,inoHeader:= THIS^.Station.CuProcessData.Header));
    //-------------------------------------
END_IF
END_METHOD

METHOD DialogExamples
VAR_INPUT
		inStepID : INT;
END_VAR
IF (Step(inStepID, TRUE, 'DIALOG EXAMPLE ')) THEN
//-------------------------------------
		_dialog.Show()
            .WithType(eDialogType.Question)
            .WithYesNo()
            .WithCaption('Hey')
            .WithText('Do we go ahead ');

        IF (_dialog.Answer = TcoCore.eDialogAnswer.Yes) THEN
            CompleteStep();
        END_IF;

        IF (_dialog.Answer = TcoCore.eDialogAnswer.No) THEN
            ;
        END_IF;

//-------------------------------------
END_IF;

IF (Step(inStepID+10, TRUE, 'DIALOG EXAMPLE WIT IMAGE')) THEN
//-------------------------------------
		_dialog.Show()
            .WithType(eDialogType.Question)
            .WithYesNo()
			.WithImage('D:\MTS\Develop\TcOpenGroup\TcOpen\assets\logo\TcOpenLogo.png',400,600)
            .WithCaption('Hey 1')
            .WithText('Do we go ahead ?');

        IF (_dialog.Answer = TcoCore.eDialogAnswer.Yes) THEN
            CompleteStep();
        END_IF;

        IF (_dialog.Answer = TcoCore.eDialogAnswer.No) THEN
            ;
        END_IF;

//-------------------------------------
END_IF;


IF (Step(inStepID+20, TRUE, 'DIALOG EXAMPLE WITH CLOSE FROM PLC')) THEN
//-------------------------------------
		_dialog.ShowWithExternalClose(inOkAnswerSignal:=FALSE , inYesAnswerSignal:= CurrentStep.Duration>T#2000MS, inNoAnswerSignal:= FALSE, inCancelAnswerSignal:= FALSE)
		    .WithType(eDialogType.Info)
            .WithYesNoCancel()
            .WithCaption('Hey')
            .WithText('Do you wana retry it? Yes answer will be set in 4 sec?');

        IF (_dialog.Answer = TcoCore.eDialogAnswer.Yes) THEN
            CompleteStep();
        END_IF;

      

//-------------------------------------
END_IF;

IF (Step(inStepID+30, TRUE, 'CUSTOMIZED DIALOG EXAMPLE WITH CLOSE FROM PLC ')) THEN
//-------------------------------------
			 _dialogCustomized.ShowWithExternalClose(inOption1AnswerSignal:=FALSE,inOption2AnswerSignal:=FALSE, inOption3AnswerSignal:=CurrentStep.Duration>T#4000MS,inOption4AnswerSignal:=FALSE)
            
            .WithOption1('This is Option1=>retry')
			  .WithOption2('This is Option2=>first step')
			    .WithOption3('This is Option3 =>continue and finish in 4s')
			.WithImage('D:\MTS\Develop\TcOpenGroup\TcOpen\assets\logo\TcOpenWide.png',500,500)
            .WithCaption('Hey')
            .WithText('What we are going to do.');
            
		
           
	
			IF (_dialogCustomized.Answer = TcoCore.eCustomizedDialogAnswer.Option3) THEN
				CompleteStep();
			END_IF;

//-------------------------------------
END_IF;

IF (Step(inStepID+40, TRUE, 'INPUT DIALOG EXAMPLE  REQURED FIELDS TO INPUT DATA')) THEN
//-------------------------------------
		_dialogWithInput.Show(refContent:=_customizedContentInput)
            .WithType(eDialogType.Question)
            .WithYesNo()
            .WithCaption('Hey wana set data')
            .WithText('Do you realy want to sent data to ....?');
                
		IF (_dialogWithInput.Answer = TcoCore.eInputDialogAnswer.Yes) THEN
				CompleteStep();
			//by yes or (ok) option data are confirmed and transfered to plc (_customizedContentInput)
		ELSIF (_dialogWithInput.Answer = TcoCore.eInputDialogAnswer.No) THEN
			// data in struct '_customizedContentInput' remains same as before
 		END_IF;
		

//-------------------------------------
END_IF;
IF (Step(inStepID+50, TRUE, 'INPUT DIALOG EXAMPLE WITH WEB CONTENT AND REQURED FIELDS TO INPUT DATA')) THEN
//-------------------------------------
		_dialogWithInput.Show(refContent:=_customizedContentInput)
            .WithType(eDialogType.Question)
            .WithOk()
			.WithImage('https://github.com/TcOpenGroup',400,600)
            .WithCaption('Hey wana set data')
            .WithText('Do you realy want to sent data to ....?');
			
                
		IF (_dialogWithInput.Answer = TcoCore.eInputDialogAnswer.OK) THEN
			CompleteStep();
			
		END_IF;

//-------------------------------------
END_IF;
END_METHOD

METHOD GroupedExample
VAR_INPUT
		inStepID : INT;
END_VAR
IF (Step(inStepID, TRUE, 'MULTI ANALOGUE INSPECTIONS PART 1 WITH WEB CONTENT')) THEN
//-------------------------------------
		Station.GroupInspection
		.WithCoordinator(THIS^)
		.Act();
		Station.GroupInspection.Inspect(Station.ProcessDataManager.Data.CU00x.Dim_Inspector_1.WithCoordinator(THIS^).Inspect(0));	
		Station.GroupInspection.Inspect(Station.ProcessDataManager.Data.CU00x.Dim_Inspector_2.WithCoordinator(THIS^).Inspect(0));	
		Station.GroupInspection.Inspect(Station.ProcessDataManager.Data.CU00x.Dim_Inspector_3.WithCoordinator(THIS^).Inspect(0));	
		Station.GroupInspection.Inspect(Station.ProcessDataManager.Data.CU00x.Dim_Inspector_4.WithCoordinator(THIS^).Inspect(0));	
		Station.GroupInspection.Inspect(Station.ProcessDataManager.Data.CU00x.Dim_Inspector_5.WithCoordinator(THIS^).Inspect(0));	
		Station.GroupInspection.Inspect(Station.ProcessDataManager.Data.CU00x.Dim_Inspector_6.WithCoordinator(THIS^).Inspect(1));	
		Station.GroupInspection.Inspect(Station.ProcessDataManager.Data.CU00x.Dim_Inspector_7.WithCoordinator(THIS^).Inspect(0));	
		Station.GroupInspection.Inspect(Station.ProcessDataManager.Data.CU00x.Dim_Inspector_8.WithCoordinator(THIS^).Inspect(0));	
		Station.GroupInspection.Inspect(Station.ProcessDataManager.Data.CU00x.Dim_Inspector_9.WithCoordinator(THIS^).Inspect(0));	
		Station.GroupInspection.Inspect(Station.ProcessDataManager.Data.CU00x.Dim_Inspector_10.WithCoordinator(THIS^).Inspect(0));	
	
		
		Station.GroupInspection.UpdateComprehensiveResult(Station.ProcessDataManager.Data.EntityHeader.Results)	
		.Instruct('Something is wrong 1')
		.InstructWithImage('https://github.com/TcOpenGroup/TcOpen/blob/dev/README.md',400,600)	
		.OnFail()
		.Dialog(inStepID+10);			
//-------------------------------------
END_IF;

IF (Step(inStepID+10, TRUE, 'MULTI ANALOGUE INSPECTIONS PART 2 WITH INSTRUCTION AND DESCRIPTION')) THEN
//-------------------------------------
		Station.GroupInspection
		.WithCoordinator(THIS^)
		.Act();
		Station.GroupInspection.Inspect(Station.ProcessDataManager.Data.CU00x.Dim_Inspector_11.WithCoordinator(THIS^).Inspect(0));	
		Station.GroupInspection.Inspect(Station.ProcessDataManager.Data.CU00x.Dim_Inspector_12.WithCoordinator(THIS^).Inspect(0));	
		Station.GroupInspection.Inspect(Station.ProcessDataManager.Data.CU00x.Dim_Inspector_13.WithCoordinator(THIS^).Inspect(0));	
		Station.GroupInspection.Inspect(Station.ProcessDataManager.Data.CU00x.Dim_Inspector_14.WithCoordinator(THIS^).Inspect(0));	
		Station.GroupInspection.Inspect(Station.ProcessDataManager.Data.CU00x.Dim_Inspector_15.WithCoordinator(THIS^).Inspect(0));	
		Station.GroupInspection.Inspect(Station.ProcessDataManager.Data.CU00x.Dim_Inspector_16.WithCoordinator(THIS^).Inspect(1));	
		Station.GroupInspection.Inspect(Station.ProcessDataManager.Data.CU00x.Dim_Inspector_17.WithCoordinator(THIS^).Inspect(0));	
		Station.GroupInspection.Inspect(Station.ProcessDataManager.Data.CU00x.Dim_Inspector_18.WithCoordinator(THIS^).Inspect(0));	
		Station.GroupInspection.Inspect(Station.ProcessDataManager.Data.CU00x.Dim_Inspector_19.WithCoordinator(THIS^).Inspect(0));	
		Station.GroupInspection.Inspect(Station.ProcessDataManager.Data.CU00x.Dim_Inspector_20.WithCoordinator(THIS^).Inspect(0));	
	
		
		Station.GroupInspection.UpdateComprehensiveResult(Station.ProcessDataManager.Data.EntityHeader.Results)	
		.WithDescription()
		.Instruct('Something is wrong 2')
		.OnFail()
		.Dialog(inStepID+20);			
//-------------------------------------
END_IF;



IF (Step(inStepID+20, TRUE, 'MULTI ANALOGUE INSPECTIONS PART 2 WITH INSTRUCTION AND DESCRIPTION EVAVLUATED')) THEN
//-------------------------------------

		Station.GroupInspection
		.WithCoordinator(THIS^)
		.Act();
		Station.GroupInspection.Inspect(Station.ProcessDataManager.Data.CU00x.Dim_Inspector_11.WithCoordinator(THIS^).Inspect(0));	
		Station.GroupInspection.Inspect(Station.ProcessDataManager.Data.CU00x.Dim_Inspector_12.WithCoordinator(THIS^).Inspect(0));	
		Station.GroupInspection.Inspect(Station.ProcessDataManager.Data.CU00x.Dim_Inspector_13.WithCoordinator(THIS^).Inspect(0));	
		Station.GroupInspection.Inspect(Station.ProcessDataManager.Data.CU00x.Dim_Inspector_14.WithCoordinator(THIS^).Inspect(0));	
		Station.GroupInspection.Inspect(Station.ProcessDataManager.Data.CU00x.Dim_Inspector_15.WithCoordinator(THIS^).Inspect(0));	
		Station.GroupInspection.Inspect(Station.ProcessDataManager.Data.CU00x.Dim_Inspector_16.WithCoordinator(THIS^).Inspect(1));	
		Station.GroupInspection.Inspect(Station.ProcessDataManager.Data.CU00x.Dim_Inspector_17.WithCoordinator(THIS^).Inspect(0));	
		Station.GroupInspection.Inspect(Station.ProcessDataManager.Data.CU00x.Dim_Inspector_18.WithCoordinator(THIS^).Inspect(0));	
		Station.GroupInspection.Inspect(Station.ProcessDataManager.Data.CU00x.Dim_Inspector_19.WithCoordinator(THIS^).Inspect(0));	
		Station.GroupInspection.Inspect(Station.ProcessDataManager.Data.CU00x.Dim_Inspector_20.WithCoordinator(THIS^).Inspect(0));	
	
		
		Station.GroupInspection.UpdateComprehensiveResult(Station.ProcessDataManager.Data.EntityHeader.Results)	
		.WithDescription()
		.Instruct('Something is wrong')
		.OnFail().Evaluate(	inStepID+10,eTcoInspectorFailMode.RetryThenCarryOn,inStepId+30);
//-------------------------------------
END_IF;

IF (Step(inStepID+30, TRUE, 'DONE')) THEN
//-------------------------------------
		CompleteStep();
//-------------------------------------
END_IF;
END_METHOD

(*~
	<docu>
		<summary>
			Main method of the sequener. Custom code needs to be placed here. The sequencer is executed by call of **Instance.Run()** method.
			This method is abstract, and it must be overridden in derived block.
		</summary>
	</docu>
~*)
METHOD PROTECTED Main : BOOL
(*

	OPENING DATA OPERATIONS
	Following methods provide process data manipulation for this controlled unit.
	Remove `IF` statement and comment or uncomment according to your need.
*)
// Loads process settings. 
// Typically used in the first station of the technology to load process settings that will be used trough out the production
IF (_dataLoadProcessSettings) THEN
    THIS^.DataLoadProcessSettings(100);
END_IF;

// Loads process settings via produciton planer. 
// Typically used in the first station of the technology to load process settings that will be used trough out the production 
// .......
IF (_dataLoadProcessSettingsByPlaner) THEN
    THIS^.DataLoadProcessSettingsByPlaner(110);
END_IF;

(*

		
		This step we would like to star cycle time (e.g. we want to exclude loading data from clean cycle time )		
*)
IF (Step(150, TRUE, '<#START MEASURE CT TRIGGER#>')) THEN
    //-------------------------------------    
    StartCleanCycleTime();

	CustomObserver.DefineControledUnit(THIS^.Station.CuId);
	
    StepCompleteWhen(TRUE);
    //-------------------------------------
END_IF

// Creates new data entity (new part/item) 
// Typically used in the first station of the technology to create new document/record to be persited in the repository.
// Sets the status of the entity to 'InProgress'
IF (_dataCreateNew) THEN
	IF (Step(160, TRUE, 'CREATE ENTIY ID')) THEN
		//-------------------------------------    
		Station.ProcessDataManager.Data._EntityId := ULINT_TO_STRING(Context.RealTimeClock.TickClock());
	
		StepCompleteWhen(Station.ProcessDataManager.Data._EntityId<>'');
		//-------------------------------------
	END_IF
    THIS^.DataEntityCreateNew(200, Station.ProcessDataManager.Data._EntityId, Header := Station.ProcessDataManager.Data.CU00x.Header);
END_IF;

// Populates the information in the data header of this controlled unit (operation start time stamp, user info, etc)
// Typically used prior to starting operation within a controlled unit.
IF (_dataOpen) THEN
    THIS^.DataEntityOpen(300,
        30000,
        Station.ProcessDataManager.Data._EntityId,
        Station.ProcessDataManager.Data.CU00x.Header);
END_IF;


// Handle user defined carier id
// Typically used in the first station of the technology to assign user defined carier ID  instead of raw unique id(RfidChip....)
IF (_tagsPairing) THEN
    THIS^.PairTag(400);
END_IF;
(*

		STEPS OF THE SEQUENCE
		Here we would place steps to perfom the operations of this controlled unit.

*)



IF (Step(900, TRUE, 'SINGLE INSPECTION')) THEN
    //-------------------------------------    
	Station.ProcessDataManager.Data.CU00x.BoltPresenceInspector.Data.FailureDescription:='BoltPresenceInspector error';
    Station.ProcessDataManager.Data.CU00x.BoltPresenceInspector.WithCoordinator(THIS^)
        .Inspect(_inspectionResult)
        .UpdateComprehensiveResult(Station.ProcessDataManager.Data.EntityHeader.Results)
        .OnFail().CarryOn();
    //-------------------------------------
END_IF

IF (Step(910, TRUE, 'SINGLE ANALOGUE INSPECTION')) THEN
    //-------------------------------------    
		Station.ProcessDataManager.Data.CU00x.BoltDimensionPresenceInspector.Data.FailureDescription:='BoltDimensionPresenceInspector error';

    Station.ProcessDataManager.Data.CU00x.BoltDimensionPresenceInspector.WithCoordinator(THIS^)
        .Inspect(_inspectionDimensionResult)
        .UpdateComprehensiveResult(Station.ProcessDataManager.Data.EntityHeader.Results)
        .OnFail().Dialog(300);
    //-------------------------------------
END_IF


//dialog usage examples
IF _dialogExamples THEN
	DialogExamples(1000);
END_IF;

//single inspexction usage
IF _inspectorSingleExamples THEN
	SingleExample(1100);
END_IF;

// grouped usage of isnpectors
IF _inspectorGroupExamples THEN
	GroupedExample(1200);
END_IF;


IF (Step(2000, true, 'START PARALELL TASK')) THEN
    //-------------------------------------    
    StepCompleteWhen(_paralellTask.Task.Invoke().Busy);
    //-------------------------------------
END_IF

(*

		RECOVERY STEPS
		This step and the following steps should bring the controlled unit in a state from which 
		the sequence can be safely restarted from the beginning of the this sequencer. 		
*)
IF (Step(RESTORE_STEP_ID, TRUE, 'FIRST RESTORE STEP')) THEN
    //-------------------------------------
    StepCompleteWhen(_continueRestore);
    //-------------------------------------	
END_IF

(*

		
